_i:=E_Cylinder.OpenLockPush;
G_arrCylinder[_i].stInput.bHome:=GVL.I.bOpenLockPush_Cyl_H;
G_arrCylinder[_i].stInput.bWork:=GVL.I.bOpenLockPush_Cyl_W;
GVL.Q.bOpenLockPush_Cyl_H:=G_arrCylinder[_i].stOutput.bHome;
GVL.Q.bOpenLockPush_Cyl_W:=G_arrCylinder[_i].stOutput.bWork;

_i:=E_Cylinder.OpenLockRotate;
G_arrCylinder[_i].stInput.bHome:=GVL.I.bOpenLockRotate_Cyl_H;
G_arrCylinder[_i].stInput.bWork:=GVL.I.bOpenLockRotate_Cyl_W;
GVL.Q.bOpenLockRotate_Cyl_H:=G_arrCylinder[_i].stOutput.bHome;
GVL.Q.bOpenLockRotate_Cyl_W:=G_arrCylinder[_i].stOutput.bWork;

_i:=E_Cylinder.OpenLockPush2;
//G_arrCylinder[_i].stInput.bHome:=GVL.I.bOpenLockPush2_Cyl_H;
G_arrCylinder[_i].stInput.bHome:=NOT GVL.I.bOpenLockPush2_Cyl_W;
G_arrCylinder[_i].stInput.bWork:=GVL.I.bOpenLockPush2_Cyl_W;
GVL.Q.bOpenLockPush2_Cyl_H:=G_arrCylinder[_i].stOutput.bHome;
GVL.Q.bOpenLockPush2_Cyl_W:=G_arrCylinder[_i].stOutput.bWork;

_i:=E_Cylinder.TakeUcPrevent;
G_arrCylinder[_i].stInput.bWork:=GVL.I.bTakeUcPrevent_Cyl_W;
GVL.Q.bTakeUcPrevent_Cyl_H:=G_arrCylinder[_i].stOutput.bHome;
GVL.Q.bTakeUcPrevent_Cyl_W:=G_arrCylinder[_i].stOutput.bWork;

_i:=E_Cylinder.TakeUcLift;
G_arrCylinder[_i].stInput.bHome:=GVL.I.bTakeUcLift_Cyl_H;
G_arrCylinder[_i].stInput.bWork:=G_arrCylinder[_i].stOutput.bWork;//GVL.I.bTakeUcLift_Cyl_W;
GVL.Q.bTakeUcLift_Cyl_H:=G_arrCylinder[_i].stOutput.bHome;
GVL.Q.bTakeUcLift_Cyl_W:=G_arrCylinder[_i].stOutput.bWork;

_i:=E_Cylinder.TakeUcPush;
G_arrCylinder[_i].stInput.bHome:=GVL.I.bTakeUcPush_Cyl_H;
G_arrCylinder[_i].stInput.bWork:=GVL.I.bTakeUcPush_Cyl_W;
GVL.Q.bTakeUcPush_Cyl_H:=G_arrCylinder[_i].stOutput.bHome;
GVL.Q.bTakeUcPush_Cyl_W:=G_arrCylinder[_i].stOutput.bWork;

_i:=E_Cylinder.TakeUcRotate;
G_arrCylinder[_i].stInput.bHome:=GVL.I.bTakeUcRotate_Cyl_H;
G_arrCylinder[_i].stInput.bWork:=GVL.I.bTakeUcRotate_Cyl_W;
GVL.Q.bTakeUcRotate_Cyl_H:=G_arrCylinder[_i].stOutput.bHome;
GVL.Q.bTakeUcRotate_Cyl_W:=G_arrCylinder[_i].stOutput.bWork;

_i:=E_Cylinder.TakeUcStandard;
G_arrCylinder[_i].stInput.bHome:=GVL.I.bTakeUcStandard_Cyl_H;
G_arrCylinder[_i].stInput.bWork:=GVL.I.bTakeUcStandard_Cyl_W;
GVL.Q.bTakeUcStandard_Cyl_H:=G_arrCylinder[_i].stOutput.bHome;
GVL.Q.bTakeUcStandard_Cyl_W:=G_arrCylinder[_i].stOutput.bWork;

_i:=E_Cylinder.UnloadFrockPrevent;
G_arrCylinder[_i].stInput.bHome:=GVL.I.bUnloadFrockPrevent_Cyl_H;
G_arrCylinder[_i].stInput.bWork:=GVL.I.bUnloadFrockPrevent_Cyl_W;
GVL.Q.bUnloadFrockPrevent_Cyl_H:=G_arrCylinder[_i].stOutput.bHome;
GVL.Q.bUnloadFrockPrevent_Cyl_W:=G_arrCylinder[_i].stOutput.bWork;

_i:=E_Cylinder.UnloadFrockLift;
G_arrCylinder[_i].stInput.bHome:=GVL.I.bUnloadFrockLift_Cyl_H;
G_arrCylinder[_i].stInput.bWork:=GVL.I.bUnloadFrockLift_Cyl_W;
GVL.Q.bUnloadFrockLift_Cyl_H:=G_arrCylinder[_i].stOutput.bHome;
GVL.Q.bUnloadFrockLift_Cyl_W:=G_arrCylinder[_i].stOutput.bWork;

_i:=E_Cylinder.UnloadFrockPush;
G_arrCylinder[_i].stInput.bHome:=GVL.I.bUnloadFrockPush_Cyl_H;
G_arrCylinder[_i].stInput.bWork:=GVL.I.bUnloadFrockPush_Cyl_W;
GVL.Q.bUnloadFrockPush_Cyl_H:=G_arrCylinder[_i].stOutput.bHome;
GVL.Q.bUnloadFrockPush_Cyl_W:=G_arrCylinder[_i].stOutput.bWork;

_i:=E_Cylinder.TakeUc1Y;
G_arrCylinder[_i].stInput.bHome:=GVL.I.bTakeUc1Y_Cyl_H;
G_arrCylinder[_i].stInput.bWork:=GVL.I.bTakeUc1Y_Cyl_W;
GVL.Q.bTakeUc1Y_Cyl_H:=G_arrCylinder[_i].stOutput.bHome;
GVL.Q.bTakeUc1Y_Cyl_W:=G_arrCylinder[_i].stOutput.bWork;

_i:=E_Cylinder.TakeUc1Z1;
G_arrCylinder[_i].stInput.bHome:=GVL.I.bTakeUc1Z1_Cyl_H;
G_arrCylinder[_i].stInput.bWork:=GVL.I.bTakeUc1Z1_Cyl_W;
GVL.Q.bTakeUc1Z1_Cyl_H:=G_arrCylinder[_i].stOutput.bHome;
GVL.Q.bTakeUc1Z1_Cyl_W:=G_arrCylinder[_i].stOutput.bWork;

_i:=E_Cylinder.TakeUc1Z2;
G_arrCylinder[_i].stInput.bHome:=GVL.I.bTakeUc1Z2_Cyl_H;
G_arrCylinder[_i].stInput.bWork:=GVL.I.bTakeUc1Z2_Cyl_W;
GVL.Q.bTakeUc1Z2_Cyl_H:=G_arrCylinder[_i].stOutput.bHome;
GVL.Q.bTakeUc1Z2_Cyl_W:=G_arrCylinder[_i].stOutput.bWork;

_i:=E_Cylinder.TakeUc1Rotate;
G_arrCylinder[_i].stInput.bHome:=GVL.I.bTakeUc1Rotate_Cyl_H;
G_arrCylinder[_i].stInput.bWork:=GVL.I.bTakeUc1Rotate_Cyl_W;
GVL.Q.bTakeUc1Rotate_Cyl_H:=G_arrCylinder[_i].stOutput.bHome;
GVL.Q.bTakeUc1Rotate_Cyl_W:=G_arrCylinder[_i].stOutput.bWork;

_i:=E_Cylinder.TakeUc1Clamp;
G_arrCylinder[_i].stInput.bHome:=GVL.I.bTakeUc1Clamp_Cyl_H;
//G_arrCylinder[_i].stInput.bWork:=GVL.I.bTakeUc1Clamp_Cyl_W;
GVL.Q.bTakeUc1Clamp_Cyl_H:=G_arrCylinder[_i].stOutput.bHome;
GVL.Q.bTakeUc1Clamp_Cyl_W:=G_arrCylinder[_i].stOutput.bWork;

_i:=E_Cylinder.UnloadUcElevator;
//G_arrCylinder[_i].stInput.bHome:=GVL.I.bUnloadUcElevator_Cyl_H;
//G_arrCylinder[_i].stInput.bWork:=GVL.I.bUnloadUcElevator_Cyl_W;
GVL.Q.bUnloadUcElevator_Cyl_H:=G_arrCylinder[_i].stOutput.bHome;
GVL.Q.bUnloadUcElevator_Cyl_W:=G_arrCylinder[_i].stOutput.bWork;

_i:=E_Cylinder.UnloadUcConveyorPush;
//G_arrCylinder[_i].stInput.bHome:=GVL.I.bUnloadUcConveyorPush_Cyl_H;
//G_arrCylinder[_i].stInput.bWork:=GVL.I.bUnloadUcConveyorPush_Cyl_W;
GVL.Q.bUnloadUcConveyorPush_Cyl_H:=G_arrCylinder[_i].stOutput.bHome;
GVL.Q.bUnloadUcConveyorPush_Cyl_W:=G_arrCylinder[_i].stOutput.bWork;

_i:=E_Cylinder.UnloadFrockConveyorPrevent;
//G_arrCylinder[_i].stInput.bHome:=GVL.I.bUnloadFrockConveyorPrevent_Cyl_H;
//G_arrCylinder[_i].stInput.bWork:=GVL.I.bUnloadFrockConveyorPrevent_Cyl_W;
GVL.Q.bUnloadFrockConveyorPrevent_Cyl_H:=G_arrCylinder[_i].stOutput.bHome;
GVL.Q.bUnloadFrockConveyorPrevent_Cyl_W:=G_arrCylinder[_i].stOutput.bWork;

_i:=E_Cylinder.UnloadFrockConveyorPush;
//G_arrCylinder[_i].stInput.bHome:=GVL.I.bUnloadFrockConveyorPush_Cyl_H;
//G_arrCylinder[_i].stInput.bWork:=GVL.I.bUnloadFrockConveyorPush_Cyl_W;
GVL.Q.bUnloadFrockConveyorPush_Cyl_H:=G_arrCylinder[_i].stOutput.bHome;
GVL.Q.bUnloadFrockConveyorPush_Cyl_W:=G_arrCylinder[_i].stOutput.bWork;

_i:=E_Cylinder.OpenLockElevator;
G_arrCylinder[_i].stInput.bHome:=GVL.I.bOpenLockElevator_Cyl_H;
G_arrCylinder[_i].stInput.bWork:=GVL.I.bOpenLockElevator_Cyl_W;
GVL.Q.bOpenLockElevator_Cyl_H:=G_arrCylinder[_i].stOutput.bHome;
GVL.Q.bOpenLockElevator_Cyl_W:=G_arrCylinder[_i].stOutput.bWork;

_i:=E_Cylinder.OpenLockPin;
G_arrCylinder[_i].stInput.bWork:=G_arrCylinder[_i].stOutput.bWork;//GVL.I.bOpenLockPin_Cyl_W;
GVL.Q.bOpenLockPin_Cyl_H:=G_arrCylinder[_i].stOutput.bHome;
GVL.Q.bOpenLockPin_Cyl_W:=G_arrCylinder[_i].stOutput.bWork;

_i:=E_Cylinder.TakeUcElevator;
G_arrCylinder[_i].stInput.bHome:=GVL.I.bTakeUcElevator_Cyl_H;
G_arrCylinder[_i].stInput.bWork:=GVL.I.bTakeUcElevator_Cyl_W;
GVL.Q.bTakeUcElevator_Cyl_H:=G_arrCylinder[_i].stOutput.bHome;
GVL.Q.bTakeUcElevator_Cyl_W:=G_arrCylinder[_i].stOutput.bWork;

_i:=E_Cylinder.TakeUcPush1;
G_arrCylinder[_i].stInput.bHome:=GVL.I.bTakeUcPush1_Cyl_H;
G_arrCylinder[_i].stInput.bWork:=GVL.I.bTakeUcPush1_Cyl_W;
GVL.Q.bTakeUcPush1_Cyl_H:=G_arrCylinder[_i].stOutput.bHome;
GVL.Q.bTakeUcPush1_Cyl_W:=G_arrCylinder[_i].stOutput.bWork;

_i:=E_Cylinder.UnloadUcBeltTipper;
G_arrCylinder[_i].stInput.bHome:=GVL.I.bUnloadUcBeltTipper_Cyl_H;
G_arrCylinder[_i].stInput.bWork:=GVL.I.bUnloadUcBeltTipper_Cyl_W;
GVL.Q.bUnloadUcBeltTipper_Cyl_H:=G_arrCylinder[_i].stOutput.bHome;
GVL.Q.bUnloadUcBeltTipper_Cyl_W:=G_arrCylinder[_i].stOutput.bWork;

_i:=E_Cylinder.UnloadUcBeltLift;
G_arrCylinder[_i].stInput.bHome:=GVL.I.bUnloadUcBeltLift_Cyl_H;
G_arrCylinder[_i].stInput.bWork:=GVL.I.bUnloadUcBeltLift_Cyl_W;
GVL.Q.bUnloadUcBeltLift_Cyl_H:=G_arrCylinder[_i].stOutput.bHome;
GVL.Q.bUnloadUcBeltLift_Cyl_W:=G_arrCylinder[_i].stOutput.bWork;

_i:=E_Cylinder.OpenLockTranslation;
G_arrCylinder[_i].stInput.bHome:=GVL.I.bOpenLockTranslation_Cyl_H;
G_arrCylinder[_i].stInput.bWork:=GVL.I.bOpenLockTranslation_Cyl_W;
GVL.Q.bOpenLockTranslation_Cyl_H:=G_arrCylinder[_i].stOutput.bHome;
GVL.Q.bOpenLockTranslation_Cyl_W:=G_arrCylinder[_i].stOutput.bWork;

_i:=E_Cylinder.TakeUcFrockClamp;
G_arrCylinder[_i].stInput.bHome:=GVL.I.bTakeUcFrockClamp_Cyl_H;
G_arrCylinder[_i].stInput.bWork:=GVL.I.bTakeUcFrockClamp_Cyl_W;
GVL.Q.bTakeUcFrockClamp_Cyl_H:=G_arrCylinder[_i].stOutput.bHome;
GVL.Q.bTakeUcFrockClamp_Cyl_W:=G_arrCylinder[_i].stOutput.bWork;
END_ACTION

ACTION A_CylinderTest367:
FOR _i:=0 TO 50 BY 1 DO
	G_arrCylinder[_i].ID:=TO_BYTE(_i+50);
	_arrCylTon_H[_i](IN:=G_arrCylinder[_i].stOutput.bHome , PT:=T#2S , Q=> , ET=> );
	_arrCylTon_W[_i](IN:=G_arrCylinder[_i].stOutput.bWork , PT:=T#2S , Q=> , ET=> );
	G_arrCylinder[_i].stInput.bHome:=_arrCylTon_H[_i].Q;
	G_arrCylinder[_i].stInput.bWork:=_arrCylTon_W[_i].Q;
END_FOR

_i:=E_Cylinder.Line0Part;
GVL.Q.bLine0Part_Cyl_H:=G_arrCylinder[_i].stOutput.bHome;
GVL.Q.bLine0Part_Cyl_W:=G_arrCylinder[_i].stOutput.bWork;

_i:=E_Cylinder.Line0Prevent;
GVL.Q.bLine0Prevent_Cyl_H:=G_arrCylinder[_i].stOutput.bHome;
GVL.Q.bLine0Prevent_Cyl_W:=G_arrCylinder[_i].stOutput.bWork;

_i:=E_Cylinder.Line0Push;
G_arrCylinder[_i].stInput.bHome:=GVL.I.bLine0Push_Cyl_H;
G_arrCylinder[_i].stInput.bWork:=GVL.I.bLine0Push_Cyl_W;
GVL.Q.bLine0Push_Cyl_H:=G_arrCylinder[_i].stOutput.bHome;
GVL.Q.bLine0Push_Cyl_W:=G_arrCylinder[_i].stOutput.bWork;

_i:=E_Cylinder.AcquirePrevent0;
G_arrCylinder[_i].stInput.bWork:=GVL.I.bAcquirePrevent0_Cyl_W;
GVL.Q.bAcquirePrevent0_Cyl_H:=G_arrCylinder[_i].stOutput.bHome;
GVL.Q.bAcquirePrevent0_Cyl_W:=G_arrCylinder[_i].stOutput.bWork;

_i:=E_Cylinder.AcquirePrevent1;
G_arrCylinder[_i].stInput.bWork:=GVL.I.bAcquirePrevent1_Cyl_W;
GVL.Q.bAcquirePrevent1_Cyl_H:=G_arrCylinder[_i].stOutput.bHome;
GVL.Q.bAcquirePrevent1_Cyl_W:=G_arrCylinder[_i].stOutput.bWork;

_i:=E_Cylinder.AcquireLift;
G_arrCylinder[_i].stInput.bHome:=GVL.I.bAcquireLift_Cyl_H;
G_arrCylinder[_i].stInput.bWork:=GVL.I.bAcquireLift_Cyl_W;
GVL.Q.bAcquireLift_Cyl_H:=G_arrCylinder[_i].stOutput.bHome;
GVL.Q.bAcquireLift_Cyl_W:=G_arrCylinder[_i].stOutput.bWork;

_i:=E_Cylinder.AcquirePush;
G_arrCylinder[_i].stInput.bHome:=GVL.I.bAcquirePush_Cyl_H;
G_arrCylinder[_i].stInput.bWork:=GVL.I.bAcquirePush_Cyl_W;
GVL.Q.bAcquirePush_Cyl_H:=G_arrCylinder[_i].stOutput.bHome;
GVL.Q.bAcquirePush_Cyl_W:=G_arrCylinder[_i].stOutput.bWork;

_i:=E_Cylinder.AcquireElevator;
G_arrCylinder[_i].stInput.bHome:=GVL.I.bAcquireElevator_Cyl_H;
G_arrCylinder[_i].stInput.bWork:=GVL.I.bAcquireElevator_Cyl_W;
GVL.Q.bAcquireElevator_Cyl_H:=G_arrCylinder[_i].stOutput.bHome;
GVL.Q.bAcquireElevator_Cyl_W:=G_arrCylinder[_i].stOutput.bWork;

_i:=E_Cylinder.SteeringLift;
G_arrCylinder[_i].stInput.bHome:=GVL.I.bSteeringLift_Cyl_H;
G_arrCylinder[_i].stInput.bWork:=GVL.I.bSteeringLift_Cyl_W;
GVL.Q.bSteeringLift_Cyl_H:=G_arrCylinder[_i].stOutput.bHome;
GVL.Q.bSteeringLift_Cyl_W:=G_arrCylinder[_i].stOutput.bWork;

_i:=E_Cylinder.SteeringAcquireElevator;
G_arrCylinder[_i].stInput.bHome:=GVL.I.bSteeringAcquireElevator_Cyl_H;
G_arrCylinder[_i].stInput.bWork:=GVL.I.bSteeringAcquireElevator_Cyl_W;
GVL.Q.bSteeringAcquireElevator_Cyl_H:=G_arrCylinder[_i].stOutput.bHome;
GVL.Q.bSteeringAcquireElevator_Cyl_W:=G_arrCylinder[_i].stOutput.bWork;

_i:=E_Cylinder.SteeringRotate;
G_arrCylinder[_i].stInput.bHome:=GVL.I.bSteeringRotate_Cyl_H;
G_arrCylinder[_i].stInput.bWork:=GVL.I.bSteeringRotate_Cyl_W;
GVL.Q.bSteeringRotate_Cyl_H:=G_arrCylinder[_i].stOutput.bHome;
GVL.Q.bSteeringRotate_Cyl_W:=G_arrCylinder[_i].stOutput.bWork;

_i:=E_Cylinder.SteeringAcquireLimit;
G_arrCylinder[_i].stInput.bHome:=GVL.I.bSteeringAcquireLimit_Cyl_H;
G_arrCylinder[_i].stInput.bWork:=GVL.I.bSteeringAcquireLimit_Cyl_W;
GVL.Q.bSteeringAcquireLimit_Cyl_H:=G_arrCylinder[_i].stOutput.bHome;
GVL.Q.bSteeringAcquireLimit_Cyl_W:=G_arrCylinder[_i].stOutput.bWork;

_i:=E_Cylinder.OpenLockPrevent;
G_arrCylinder[_i].stInput.bWork:=GVL.I.bOpenLockPrevent_Cyl_W;
GVL.Q.bOpenLockPrevent_Cyl_H:=G_arrCylinder[_i].stOutput.bHome;
GVL.Q.bOpenLockPrevent_Cyl_W:=G_arrCylinder[_i].stOutput.bWork;

_i:=E_Cylinder.OpenLockLift;
G_arrCylinder[_i].stInput.bHome:=GVL.I.bOpenLockLift_Cyl_H;
G_arrCylinder[_i].stInput.bWork:=GVL.I.bOpenLockLift_Cyl_W;
GVL.Q.bOpenLockLift_Cyl_H:=G_arrCylinder[_i].stOutput.bHome;
GVL.Q.bOpenLockLift_Cyl_W:=G_arrCylinder[_i].stOutput.bWork;

_i:=E_Cylinder.OpenLockPush;
G_arrCylinder[_i].stInput.bHome:=GVL.I.bOpenLockPush_Cyl_H;
G_arrCylinder[_i].stInput.bWork:=GVL.I.bOpenLockPush_Cyl_W;
GVL.Q.bOpenLockPush_Cyl_H:=G_arrCylinder[_i].stOutput.bHome;
GVL.Q.bOpenLockPush_Cyl_W:=G_arrCylinder[_i].stOutput.bWork;

_i:=E_Cylinder.OpenLockRotate;
G_arrCylinder[_i].stInput.bHome:=GVL.I.bOpenLockRotate_Cyl_H;
G_arrCylinder[_i].stInput.bWork:=GVL.I.bOpenLockRotate_Cyl_W;
GVL.Q.bOpenLockRotate_Cyl_H:=G_arrCylinder[_i].stOutput.bHome;
GVL.Q.bOpenLockRotate_Cyl_W:=G_arrCylinder[_i].stOutput.bWork;

_i:=E_Cylinder.OpenLockPush2;
//G_arrCylinder[_i].stInput.bHome:=GVL.I.bOpenLockPush2_Cyl_H;
G_arrCylinder[_i].stInput.bHome:=NOT GVL.I.bOpenLockPush2_Cyl_W;
G_arrCylinder[_i].stInput.bWork:=GVL.I.bOpenLockPush2_Cyl_W;
GVL.Q.bOpenLockPush2_Cyl_H:=G_arrCylinder[_i].stOutput.bHome;
GVL.Q.bOpenLockPush2_Cyl_W:=G_arrCylinder[_i].stOutput.bWork;

_i:=E_Cylinder.TakeUcPrevent;
G_arrCylinder[_i].stInput.bWork:=GVL.I.bTakeUcPrevent_Cyl_W;
GVL.Q.bTakeUcPrevent_Cyl_H:=G_arrCylinder[_i].stOutput.bHome;
GVL.Q.bTakeUcPrevent_Cyl_W:=G_arrCylinder[_i].stOutput.bWork;

_i:=E_Cylinder.TakeUcLift;
G_arrCylinder[_i].stInput.bHome:=GVL.I.bTakeUcLift_Cyl_H;
G_arrCylinder[_i].stInput.bWork:=GVL.I.bTakeUcLift_Cyl_W;
GVL.Q.bTakeUcLift_Cyl_H:=G_arrCylinder[_i].stOutput.bHome;
GVL.Q.bTakeUcLift_Cyl_W:=G_arrCylinder[_i].stOutput.bWork;

_i:=E_Cylinder.TakeUcPush;
G_arrCylinder[_i].stInput.bHome:=GVL.I.bTakeUcPush_Cyl_H;
G_arrCylinder[_i].stInput.bWork:=GVL.I.bTakeUcPush_Cyl_W;
GVL.Q.bTakeUcPush_Cyl_H:=G_arrCylinder[_i].stOutput.bHome;
GVL.Q.bTakeUcPush_Cyl_W:=G_arrCylinder[_i].stOutput.bWork;

_i:=E_Cylinder.TakeUcRotate;
G_arrCylinder[_i].stInput.bHome:=GVL.I.bTakeUcRotate_Cyl_H;
G_arrCylinder[_i].stInput.bWork:=GVL.I.bTakeUcRotate_Cyl_W;
GVL.Q.bTakeUcRotate_Cyl_H:=G_arrCylinder[_i].stOutput.bHome;
GVL.Q.bTakeUcRotate_Cyl_W:=G_arrCylinder[_i].stOutput.bWork;

_i:=E_Cylinder.TakeUcStandard;
G_arrCylinder[_i].stInput.bHome:=GVL.I.bTakeUcStandard_Cyl_H;
G_arrCylinder[_i].stInput.bWork:=GVL.I.bTakeUcStandard_Cyl_W;
GVL.Q.bTakeUcStandard_Cyl_H:=G_arrCylinder[_i].stOutput.bHome;
GVL.Q.bTakeUcStandard_Cyl_W:=G_arrCylinder[_i].stOutput.bWork;

_i:=E_Cylinder.UnloadFrockPrevent;
G_arrCylinder[_i].stInput.bHome:=GVL.I.bUnloadFrockPrevent_Cyl_H;
G_arrCylinder[_i].stInput.bWork:=GVL.I.bUnloadFrockPrevent_Cyl_W;
GVL.Q.bUnloadFrockPrevent_Cyl_H:=G_arrCylinder[_i].stOutput.bHome;
GVL.Q.bUnloadFrockPrevent_Cyl_W:=G_arrCylinder[_i].stOutput.bWork;

_i:=E_Cylinder.UnloadFrockLift;
G_arrCylinder[_i].stInput.bHome:=GVL.I.bUnloadFrockLift_Cyl_H;
G_arrCylinder[_i].stInput.bWork:=GVL.I.bUnloadFrockLift_Cyl_W;
GVL.Q.bUnloadFrockLift_Cyl_H:=G_arrCylinder[_i].stOutput.bHome;
GVL.Q.bUnloadFrockLift_Cyl_W:=G_arrCylinder[_i].stOutput.bWork;

_i:=E_Cylinder.UnloadFrockPush;
G_arrCylinder[_i].stInput.bHome:=GVL.I.bUnloadFrockPush_Cyl_H;
G_arrCylinder[_i].stInput.bWork:=GVL.I.bUnloadFrockPush_Cyl_W;
GVL.Q.bUnloadFrockPush_Cyl_H:=G_arrCylinder[_i].stOutput.bHome;
GVL.Q.bUnloadFrockPush_Cyl_W:=G_arrCylinder[_i].stOutput.bWork;

_i:=E_Cylinder.TakeUc1Y;
G_arrCylinder[_i].stInput.bHome:=GVL.I.bTakeUc1Y_Cyl_H;
G_arrCylinder[_i].stInput.bWork:=GVL.I.bTakeUc1Y_Cyl_W;
GVL.Q.bTakeUc1Y_Cyl_H:=G_arrCylinder[_i].stOutput.bHome;
GVL.Q.bTakeUc1Y_Cyl_W:=G_arrCylinder[_i].stOutput.bWork;

_i:=E_Cylinder.TakeUc1Z1;
G_arrCylinder[_i].stInput.bHome:=GVL.I.bTakeUc1Z1_Cyl_H;
G_arrCylinder[_i].stInput.bWork:=GVL.I.bTakeUc1Z1_Cyl_W;
GVL.Q.bTakeUc1Z1_Cyl_H:=G_arrCylinder[_i].stOutput.bHome;
GVL.Q.bTakeUc1Z1_Cyl_W:=G_arrCylinder[_i].stOutput.bWork;

_i:=E_Cylinder.TakeUc1Z2;
G_arrCylinder[_i].stInput.bHome:=GVL.I.bTakeUc1Z2_Cyl_H;
G_arrCylinder[_i].stInput.bWork:=GVL.I.bTakeUc1Z2_Cyl_W;
GVL.Q.bTakeUc1Z2_Cyl_H:=G_arrCylinder[_i].stOutput.bHome;
GVL.Q.bTakeUc1Z2_Cyl_W:=G_arrCylinder[_i].stOutput.bWork;

_i:=E_Cylinder.TakeUc1Rotate;
G_arrCylinder[_i].stInput.bHome:=GVL.I.bTakeUc1Rotate_Cyl_H;
G_arrCylinder[_i].stInput.bWork:=GVL.I.bTakeUc1Rotate_Cyl_W;
GVL.Q.bTakeUc1Rotate_Cyl_H:=G_arrCylinder[_i].stOutput.bHome;
GVL.Q.bTakeUc1Rotate_Cyl_W:=G_arrCylinder[_i].stOutput.bWork;

_i:=E_Cylinder.TakeUc1Clamp;
G_arrCylinder[_i].stInput.bHome:=GVL.I.bTakeUc1Clamp_Cyl_H;
//G_arrCylinder[_i].stInput.bWork:=GVL.I.bTakeUc1Clamp_Cyl_W;
GVL.Q.bTakeUc1Clamp_Cyl_H:=G_arrCylinder[_i].stOutput.bHome;
GVL.Q.bTakeUc1Clamp_Cyl_W:=G_arrCylinder[_i].stOutput.bWork;

_i:=E_Cylinder.UnloadUcElevator;
//G_arrCylinder[_i].stInput.bHome:=GVL.I.bUnloadUcElevator_Cyl_H;
//G_arrCylinder[_i].stInput.bWork:=GVL.I.bUnloadUcElevator_Cyl_W;
GVL.Q.bUnloadUcElevator_Cyl_H:=G_arrCylinder[_i].stOutput.bHome;
GVL.Q.bUnloadUcElevator_Cyl_W:=G_arrCylinder[_i].stOutput.bWork;

_i:=E_Cylinder.UnloadUcConveyorPush;
//G_arrCylinder[_i].stInput.bHome:=GVL.I.bUnloadUcConveyorPush_Cyl_H;
//G_arrCylinder[_i].stInput.bWork:=GVL.I.bUnloadUcConveyorPush_Cyl_W;
GVL.Q.bUnloadUcConveyorPush_Cyl_H:=G_arrCylinder[_i].stOutput.bHome;
GVL.Q.bUnloadUcConveyorPush_Cyl_W:=G_arrCylinder[_i].stOutput.bWork;

_i:=E_Cylinder.UnloadFrockConveyorPrevent;
//G_arrCylinder[_i].stInput.bHome:=GVL.I.bUnloadFrockConveyorPrevent_Cyl_H;
//G_arrCylinder[_i].stInput.bWork:=GVL.I.bUnloadFrockConveyorPrevent_Cyl_W;
GVL.Q.bUnloadFrockConveyorPrevent_Cyl_H:=G_arrCylinder[_i].stOutput.bHome;
GVL.Q.bUnloadFrockConveyorPrevent_Cyl_W:=G_arrCylinder[_i].stOutput.bWork;

_i:=E_Cylinder.UnloadFrockConveyorPush;
//G_arrCylinder[_i].stInput.bHome:=GVL.I.bUnloadFrockConveyorPush_Cyl_H;
//G_arrCylinder[_i].stInput.bWork:=GVL.I.bUnloadFrockConveyorPush_Cyl_W;
GVL.Q.bUnloadFrockConveyorPush_Cyl_H:=G_arrCylinder[_i].stOutput.bHome;
GVL.Q.bUnloadFrockConveyorPush_Cyl_W:=G_arrCylinder[_i].stOutput.bWork;

_i:=E_Cylinder.OpenLockElevator;
G_arrCylinder[_i].stInput.bHome:=GVL.I.bOpenLockElevator_Cyl_H;
G_arrCylinder[_i].stInput.bWork:=GVL.I.bOpenLockElevator_Cyl_W;
GVL.Q.bOpenLockElevator_Cyl_H:=G_arrCylinder[_i].stOutput.bHome;
GVL.Q.bOpenLockElevator_Cyl_W:=G_arrCylinder[_i].stOutput.bWork;

_i:=E_Cylinder.OpenLockPin;
G_arrCylinder[_i].stInput.bHome:=GVL.I.bOpenLockPin_Cyl_H;
G_arrCylinder[_i].stInput.bWork:=GVL.I.bOpenLockPin_Cyl_W;
GVL.Q.bOpenLockPin_Cyl_H:=G_arrCylinder[_i].stOutput.bHome;
GVL.Q.bOpenLockPin_Cyl_W:=G_arrCylinder[_i].stOutput.bWork;

_i:=E_Cylinder.TakeUcElevator;
G_arrCylinder[_i].stInput.bHome:=GVL.I.bTakeUcElevator_Cyl_H;
G_arrCylinder[_i].stInput.bWork:=GVL.I.bTakeUcElevator_Cyl_W;
GVL.Q.bTakeUcElevator_Cyl_H:=G_arrCylinder[_i].stOutput.bHome;
GVL.Q.bTakeUcElevator_Cyl_W:=G_arrCylinder[_i].stOutput.bWork;

_i:=E_Cylinder.TakeUcPush1;
G_arrCylinder[_i].stInput.bHome:=GVL.I.bTakeUcPush1_Cyl_H;
G_arrCylinder[_i].stInput.bWork:=GVL.I.bTakeUcPush1_Cyl_W;
GVL.Q.bTakeUcPush1_Cyl_H:=G_arrCylinder[_i].stOutput.bHome;
GVL.Q.bTakeUcPush1_Cyl_W:=G_arrCylinder[_i].stOutput.bWork;

_i:=E_Cylinder.UnloadUcBeltTipper;
G_arrCylinder[_i].stInput.bHome:=GVL.I.bUnloadUcBeltTipper_Cyl_H;
G_arrCylinder[_i].stInput.bWork:=GVL.I.bUnloadUcBeltTipper_Cyl_W;
GVL.Q.bUnloadUcBeltTipper_Cyl_H:=G_arrCylinder[_i].stOutput.bHome;
GVL.Q.bUnloadUcBeltTipper_Cyl_W:=G_arrCylinder[_i].stOutput.bWork;

_i:=E_Cylinder.UnloadUcBeltLift;
G_arrCylinder[_i].stInput.bHome:=GVL.I.bUnloadUcBeltLift_Cyl_H;
G_arrCylinder[_i].stInput.bWork:=GVL.I.bUnloadUcBeltLift_Cyl_W;
GVL.Q.bUnloadUcBeltLift_Cyl_H:=G_arrCylinder[_i].stOutput.bHome;
GVL.Q.bUnloadUcBeltLift_Cyl_W:=G_arrCylinder[_i].stOutput.bWork;

_i:=E_Cylinder.OpenLockTranslation;
G_arrCylinder[_i].stInput.bHome:=GVL.I.bOpenLockTranslation_Cyl_H;
G_arrCylinder[_i].stInput.bWork:=GVL.I.bOpenLockTranslation_Cyl_W;
GVL.Q.bOpenLockTranslation_Cyl_H:=G_arrCylinder[_i].stOutput.bHome;
GVL.Q.bOpenLockTranslation_Cyl_W:=G_arrCylinder[_i].stOutput.bWork;

_i:=E_Cylinder.TakeUcFrockClamp;
G_arrCylinder[_i].stInput.bHome:=G_arrCylinder[_i].stOutput.bHome;
G_arrCylinder[_i].stInput.bWork:=G_arrCylinder[_i].stOutput.bWork;
GVL.Q.bTakeUcFrockClamp_Cyl_H:=G_arrCylinder[_i].stOutput.bHome;
GVL.Q.bTakeUcFrockClamp_Cyl_W:=G_arrCylinder[_i].stOutput.bWork;
END_ACTION

ACTION A_CylinderTest373:
FOR _i:=0 TO 50 BY 1 DO
	G_arrCylinder[_i].ID:=TO_BYTE(_i+50);
	_arrCylTon_H[_i](IN:=G_arrCylinder[_i].stOutput.bHome , PT:=T#2S , Q=> , ET=> );
	_arrCylTon_W[_i](IN:=G_arrCylinder[_i].stOutput.bWork , PT:=T#2S , Q=> , ET=> );
	G_arrCylinder[_i].stInput.bHome:=_arrCylTon_H[_i].Q;
	G_arrCylinder[_i].stInput.bWork:=_arrCylTon_W[_i].Q;
END_FOR

_i:=E_Cylinder.Line0Part;
GVL.Q.bLine0Part_Cyl_H:=G_arrCylinder[_i].stOutput.bHome;
GVL.Q.bLine0Part_Cyl_W:=G_arrCylinder[_i].stOutput.bWork;

_i:=E_Cylinder.Line0Prevent;
GVL.Q.bLine0Prevent_Cyl_H:=G_arrCylinder[_i].stOutput.bHome;
GVL.Q.bLine0Prevent_Cyl_W:=G_arrCylinder[_i].stOutput.bWork;

_i:=E_Cylinder.Line0Push;
GVL.Q.bLine0Push_Cyl_H:=G_arrCylinder[_i].stOutput.bHome;
GVL.Q.bLine0Push_Cyl_W:=G_arrCylinder[_i].stOutput.bWork;

_i:=E_Cylinder.AcquirePrevent0;
G_arrCylinder[_i].stInput.bWork:=GVL.I.bAcquirePrevent0_Cyl_W;
GVL.Q.bAcquirePrevent0_Cyl_H:=G_arrCylinder[_i].stOutput.bHome;
GVL.Q.bAcquirePrevent0_Cyl_W:=G_arrCylinder[_i].stOutput.bWork;

_i:=E_Cylinder.AcquirePrevent1;
G_arrCylinder[_i].stInput.bWork:=GVL.I.bAcquirePrevent1_Cyl_W;
GVL.Q.bAcquirePrevent1_Cyl_H:=G_arrCylinder[_i].stOutput.bHome;
GVL.Q.bAcquirePrevent1_Cyl_W:=G_arrCylinder[_i].stOutput.bWork;

_i:=E_Cylinder.AcquireLift;
G_arrCylinder[_i].stInput.bHome:=GVL.I.bAcquireLift_Cyl_H;
G_arrCylinder[_i].stInput.bWork:=GVL.I.bAcquireLift_Cyl_W;
GVL.Q.bAcquireLift_Cyl_H:=G_arrCylinder[_i].stOutput.bHome;
GVL.Q.bAcquireLift_Cyl_W:=G_arrCylinder[_i].stOutput.bWork;

_i:=E_Cylinder.AcquirePush;
G_arrCylinder[_i].stInput.bHome:=GVL.I.bAcquirePush_Cyl_H;
G_arrCylinder[_i].stInput.bWork:=GVL.I.bAcquirePush_Cyl_W;
GVL.Q.bAcquirePush_Cyl_H:=G_arrCylinder[_i].stOutput.bHome;
GVL.Q.bAcquirePush_Cyl_W:=G_arrCylinder[_i].stOutput.bWork;

_i:=E_Cylinder.AcquireElevator;
G_arrCylinder[_i].stInput.bHome:=GVL.I.bAcquireElevator_Cyl_H;
G_arrCylinder[_i].stInput.bWork:=GVL.I.bAcquireElevator_Cyl_W;
GVL.Q.bAcquireElevator_Cyl_H:=G_arrCylinder[_i].stOutput.bHome;
GVL.Q.bAcquireElevator_Cyl_W:=G_arrCylinder[_i].stOutput.bWork;

_i:=E_Cylinder.SteeringLift;
G_arrCylinder[_i].stInput.bHome:=GVL.I.bSteeringLift_Cyl_H;
G_arrCylinder[_i].stInput.bWork:=GVL.I.bSteeringLift_Cyl_W;
GVL.Q.bSteeringLift_Cyl_H:=G_arrCylinder[_i].stOutput.bHome;
GVL.Q.bSteeringLift_Cyl_W:=G_arrCylinder[_i].stOutput.bWork;

_i:=E_Cylinder.SteeringAcquireElevator;
G_arrCylinder[_i].stInput.bHome:=GVL.I.bSteeringAcquireElevator_Cyl_H;
G_arrCylinder[_i].stInput.bWork:=GVL.I.bSteeringAcquireElevator_Cyl_W;
GVL.Q.bSteeringAcquireElevator_Cyl_H:=G_arrCylinder[_i].stOutput.bHome;
GVL.Q.bSteeringAcquireElevator_Cyl_W:=G_arrCylinder[_i].stOutput.bWork;

_i:=E_Cylinder.SteeringRotate;
G_arrCylinder[_i].stInput.bHome:=GVL.I.bSteeringRotate_Cyl_H;
G_arrCylinder[_i].stInput.bWork:=GVL.I.bSteeringRotate_Cyl_W;
GVL.Q.bSteeringRotate_Cyl_H:=G_arrCylinder[_i].stOutput.bHome;
GVL.Q.bSteeringRotate_Cyl_W:=G_arrCylinder[_i].stOutput.bWork;

_i:=E_Cylinder.SteeringAcquireLimit;
G_arrCylinder[_i].stInput.bHome:=GVL.I.bSteeringAcquireLimit_Cyl_H;
G_arrCylinder[_i].stInput.bWork:=GVL.I.bSteeringAcquireLimit_Cyl_W;
GVL.Q.bSteeringAcquireLimit_Cyl_H:=G_arrCylinder[_i].stOutput.bHome;
GVL.Q.bSteeringAcquireLimit_Cyl_W:=G_arrCylinder[_i].stOutput.bWork;

_i:=E_Cylinder.OpenLockPrevent;
G_arrCylinder[_i].stInput.bWork:=GVL.I.bOpenLockPrevent_Cyl_W;
GVL.Q.bOpenLockPrevent_Cyl_H:=G_arrCylinder[_i].stOutput.bHome;
GVL.Q.bOpenLockPrevent_Cyl_W:=G_arrCylinder[_i].stOutput.bWork;

_i:=E_Cylinder.OpenLockLift;
G_arrCylinder[_i].stInput.bHome:=GVL.I.bOpenLockLift_Cyl_H;
G_arrCylinder[_i].stInput.bWork:=GVL.I.bOpenLockLift_Cyl_W;
GVL.Q.bOpenLockLift_Cyl_H:=G_arrCylinder[_i].stOutput.bHome;
GVL.Q.bOpenLockLift_Cyl_W:=G_arrCylinder[_i].stOutput.bWork;

_i:=E_Cylinder.OpenLockPush;
G_arrCylinder[_i].stInput.bHome:=GVL.I.bOpenLockPush_Cyl_H;
G_arrCylinder[_i].stInput.bWork:=GVL.I.bOpenLockPush_Cyl_W;
GVL.Q.bOpenLockPush_Cyl_H:=G_arrCylinder[_i].stOutput.bHome;
GVL.Q.bOpenLockPush_Cyl_W:=G_arrCylinder[_i].stOutput.bWork;

_i:=E_Cylinder.OpenLockRotate;
G_arrCylinder[_i].stInput.bHome:=GVL.I.bOpenLockRotate_Cyl_H;
G_arrCylinder[_i].stInput.bWork:=GVL.I.bOpenLockRotate_Cyl_W;
GVL.Q.bOpenLockRotate_Cyl_H:=G_arrCylinder[_i].stOutput.bHome;
GVL.Q.bOpenLockRotate_Cyl_W:=G_arrCylinder[_i].stOutput.bWork;

_i:=E_Cylinder.OpenLockPush2;
//G_arrCylinder[_i].stInput.bHome:=GVL.I.bOpenLockPush2_Cyl_H;
G_arrCylinder[_i].stInput.bHome:=NOT GVL.I.bOpenLockPush2_Cyl_W;
G_arrCylinder[_i].stInput.bWork:=GVL.I.bOpenLockPush2_Cyl_W;
GVL.Q.bOpenLockPush2_Cyl_H:=G_arrCylinder[_i].stOutput.bHome;
GVL.Q.bOpenLockPush2_Cyl_W:=G_arrCylinder[_i].stOutput.bWork;

_i:=E_Cylinder.TakeUcPrevent;
G_arrCylinder[_i].stInput.bWork:=GVL.I.bTakeUcPrevent_Cyl_W;
GVL.Q.bTakeUcPrevent_Cyl_H:=G_arrCylinder[_i].stOutput.bHome;
GVL.Q.bTakeUcPrevent_Cyl_W:=G_arrCylinder[_i].stOutput.bWork;

_i:=E_Cylinder.TakeUcLift;
G_arrCylinder[_i].stInput.bHome:=GVL.I.bTakeUcLift_Cyl_H;
G_arrCylinder[_i].stInput.bWork:=GVL.I.bTakeUcLift_Cyl_W;
GVL.Q.bTakeUcLift_Cyl_H:=G_arrCylinder[_i].stOutput.bHome;
GVL.Q.bTakeUcLift_Cyl_W:=G_arrCylinder[_i].stOutput.bWork;

_i:=E_Cylinder.TakeUcPush;
G_arrCylinder[_i].stInput.bHome:=GVL.I.bTakeUcPush_Cyl_H;
G_arrCylinder[_i].stInput.bWork:=GVL.I.bTakeUcPush_Cyl_W;
GVL.Q.bTakeUcPush_Cyl_H:=G_arrCylinder[_i].stOutput.bHome;
GVL.Q.bTakeUcPush_Cyl_W:=G_arrCylinder[_i].stOutput.bWork;

_i:=E_Cylinder.TakeUcRotate;
G_arrCylinder[_i].stInput.bHome:=GVL.I.bTakeUcRotate_Cyl_H;
G_arrCylinder[_i].stInput.bWork:=GVL.I.bTakeUcRotate_Cyl_W;
GVL.Q.bTakeUcRotate_Cyl_H:=G_arrCylinder[_i].stOutput.bHome;
GVL.Q.bTakeUcRotate_Cyl_W:=G_arrCylinder[_i].stOutput.bWork;

_i:=E_Cylinder.TakeUcStandard;
//G_arrCylinder[_i].stInput.bHome:=GVL.I.bTakeUcStandard_Cyl_H;
//G_arrCylinder[_i].stInput.bWork:=GVL.I.bTakeUcStandard_Cyl_W;
GVL.Q.bTakeUcStandard_Cyl_H:=G_arrCylinder[_i].stOutput.bHome;
GVL.Q.bTakeUcStandard_Cyl_W:=G_arrCylinder[_i].stOutput.bWork;

_i:=E_Cylinder.UnloadFrockPrevent;
G_arrCylinder[_i].stInput.bHome:=GVL.I.bUnloadFrockPrevent_Cyl_H;
G_arrCylinder[_i].stInput.bWork:=GVL.I.bUnloadFrockPrevent_Cyl_W;
GVL.Q.bUnloadFrockPrevent_Cyl_H:=G_arrCylinder[_i].stOutput.bHome;
GVL.Q.bUnloadFrockPrevent_Cyl_W:=G_arrCylinder[_i].stOutput.bWork;

_i:=E_Cylinder.UnloadFrockLift;
G_arrCylinder[_i].stInput.bHome:=GVL.I.bUnloadFrockLift_Cyl_H;
G_arrCylinder[_i].stInput.bWork:=GVL.I.bUnloadFrockLift_Cyl_W;
GVL.Q.bUnloadFrockLift_Cyl_H:=G_arrCylinder[_i].stOutput.bHome;
GVL.Q.bUnloadFrockLift_Cyl_W:=G_arrCylinder[_i].stOutput.bWork;

_i:=E_Cylinder.UnloadFrockPush;
G_arrCylinder[_i].stInput.bHome:=GVL.I.bUnloadFrockPush_Cyl_H;
G_arrCylinder[_i].stInput.bWork:=GVL.I.bUnloadFrockPush_Cyl_W;
GVL.Q.bUnloadFrockPush_Cyl_H:=G_arrCylinder[_i].stOutput.bHome;
GVL.Q.bUnloadFrockPush_Cyl_W:=G_arrCylinder[_i].stOutput.bWork;

_i:=E_Cylinder.TakeUc1Y;
G_arrCylinder[_i].stInput.bHome:=GVL.I.bTakeUc1Y_Cyl_H;
G_arrCylinder[_i].stInput.bWork:=GVL.I.bTakeUc1Y_Cyl_W;
GVL.Q.bTakeUc1Y_Cyl_H:=G_arrCylinder[_i].stOutput.bHome;
GVL.Q.bTakeUc1Y_Cyl_W:=G_arrCylinder[_i].stOutput.bWork;

_i:=E_Cylinder.TakeUc1Z1;
G_arrCylinder[_i].stInput.bHome:=GVL.I.bTakeUc1Z1_Cyl_H;
G_arrCylinder[_i].stInput.bWork:=GVL.I.bTakeUc1Z1_Cyl_W;
GVL.Q.bTakeUc1Z1_Cyl_H:=G_arrCylinder[_i].stOutput.bHome;
GVL.Q.bTakeUc1Z1_Cyl_W:=G_arrCylinder[_i].stOutput.bWork;

_i:=E_Cylinder.TakeUc1Z2;
G_arrCylinder[_i].stInput.bHome:=GVL.I.bTakeUc1Z2_Cyl_H;
G_arrCylinder[_i].stInput.bWork:=GVL.I.bTakeUc1Z2_Cyl_W;
GVL.Q.bTakeUc1Z2_Cyl_H:=G_arrCylinder[_i].stOutput.bHome;
GVL.Q.bTakeUc1Z2_Cyl_W:=G_arrCylinder[_i].stOutput.bWork;

_i:=E_Cylinder.TakeUc1Rotate;
G_arrCylinder[_i].stInput.bHome:=GVL.I.bTakeUc1Rotate_Cyl_H;
G_arrCylinder[_i].stInput.bWork:=GVL.I.bTakeUc1Rotate_Cyl_W;
GVL.Q.bTakeUc1Rotate_Cyl_H:=G_arrCylinder[_i].stOutput.bHome;
GVL.Q.bTakeUc1Rotate_Cyl_W:=G_arrCylinder[_i].stOutput.bWork;

_i:=E_Cylinder.TakeUc1Clamp;
G_arrCylinder[_i].stInput.bHome:=GVL.I.bTakeUc1Clamp_Cyl_H;
//G_arrCylinder[_i].stInput.bWork:=GVL.I.bTakeUc1Clamp_Cyl_W;
GVL.Q.bTakeUc1Clamp_Cyl_H:=G_arrCylinder[_i].stOutput.bHome;
GVL.Q.bTakeUc1Clamp_Cyl_W:=G_arrCylinder[_i].stOutput.bWork;

_i:=E_Cylinder.UnloadUcElevator;
//G_arrCylinder[_i].stInput.bHome:=GVL.I.bUnloadUcElevator_Cyl_H;
//G_arrCylinder[_i].stInput.bWork:=GVL.I.bUnloadUcElevator_Cyl_W;
GVL.Q.bUnloadUcElevator_Cyl_H:=G_arrCylinder[_i].stOutput.bHome;
GVL.Q.bUnloadUcElevator_Cyl_W:=G_arrCylinder[_i].stOutput.bWork;

_i:=E_Cylinder.UnloadUcConveyorPush;
//G_arrCylinder[_i].stInput.bHome:=GVL.I.bUnloadUcConveyorPush_Cyl_H;
//G_arrCylinder[_i].stInput.bWork:=GVL.I.bUnloadUcConveyorPush_Cyl_W;
GVL.Q.bUnloadUcConveyorPush_Cyl_H:=G_arrCylinder[_i].stOutput.bHome;
GVL.Q.bUnloadUcConveyorPush_Cyl_W:=G_arrCylinder[_i].stOutput.bWork;

_i:=E_Cylinder.UnloadFrockConveyorPrevent;
//G_arrCylinder[_i].stInput.bHome:=GVL.I.bUnloadFrockConveyorPrevent_Cyl_H;
//G_arrCylinder[_i].stInput.bWork:=GVL.I.bUnloadFrockConveyorPrevent_Cyl_W;
GVL.Q.bUnloadFrockConveyorPrevent_Cyl_H:=G_arrCylinder[_i].stOutput.bHome;
GVL.Q.bUnloadFrockConveyorPrevent_Cyl_W:=G_arrCylinder[_i].stOutput.bWork;

_i:=E_Cylinder.UnloadFrockConveyorPush;
//G_arrCylinder[_i].stInput.bHome:=GVL.I.bUnloadFrockConveyorPush_Cyl_H;
//G_arrCylinder[_i].stInput.bWork:=GVL.I.bUnloadFrockConveyorPush_Cyl_W;
GVL.Q.bUnloadFrockConveyorPush_Cyl_H:=G_arrCylinder[_i].stOutput.bHome;
GVL.Q.bUnloadFrockConveyorPush_Cyl_W:=G_arrCylinder[_i].stOutput.bWork;

_i:=E_Cylinder.OpenLockElevator;
G_arrCylinder[_i].stInput.bHome:=GVL.I.bOpenLockElevator_Cyl_H;
G_arrCylinder[_i].stInput.bWork:=GVL.I.bOpenLockElevator_Cyl_W;
GVL.Q.bOpenLockElevator_Cyl_H:=G_arrCylinder[_i].stOutput.bHome;
GVL.Q.bOpenLockElevator_Cyl_W:=G_arrCylinder[_i].stOutput.bWork;

_i:=E_Cylinder.OpenLockPin;
G_arrCylinder[_i].stInput.bHome:=GVL.I.bOpenLockPin_Cyl_H;
G_arrCylinder[_i].stInput.bWork:=GVL.I.bOpenLockPin_Cyl_W;
GVL.Q.bOpenLockPin_Cyl_H:=G_arrCylinder[_i].stOutput.bHome;
GVL.Q.bOpenLockPin_Cyl_W:=G_arrCylinder[_i].stOutput.bWork;

_i:=E_Cylinder.TakeUcElevator;
G_arrCylinder[_i].stInput.bHome:=GVL.I.bTakeUcElevator_Cyl_H;
G_arrCylinder[_i].stInput.bWork:=GVL.I.bTakeUcElevator_Cyl_W;
GVL.Q.bTakeUcElevator_Cyl_H:=G_arrCylinder[_i].stOutput.bHome;
GVL.Q.bTakeUcElevator_Cyl_W:=G_arrCylinder[_i].stOutput.bWork;

_i:=E_Cylinder.TakeUcPush1;
G_arrCylinder[_i].stInput.bHome:=GVL.I.bTakeUcPush1_Cyl_H;
G_arrCylinder[_i].stInput.bWork:=GVL.I.bTakeUcPush1_Cyl_W;
GVL.Q.bTakeUcPush1_Cyl_H:=G_arrCylinder[_i].stOutput.bHome;
GVL.Q.bTakeUcPush1_Cyl_W:=G_arrCylinder[_i].stOutput.bWork;

_i:=E_Cylinder.UnloadUcBeltTipper;
G_arrCylinder[_i].stInput.bHome:=GVL.I.bUnloadUcBeltTipper_Cyl_H;
G_arrCylinder[_i].stInput.bWork:=GVL.I.bUnloadUcBeltTipper_Cyl_W;
GVL.Q.bUnloadUcBeltTipper_Cyl_H:=G_arrCylinder[_i].stOutput.bHome;
GVL.Q.bUnloadUcBeltTipper_Cyl_W:=G_arrCylinder[_i].stOutput.bWork;

_i:=E_Cylinder.UnloadUcBeltLift;
G_arrCylinder[_i].stInput.bHome:=GVL.I.bUnloadUcBeltLift_Cyl_H;
G_arrCylinder[_i].stInput.bWork:=GVL.I.bUnloadUcBeltLift_Cyl_W;
GVL.Q.bUnloadUcBeltLift_Cyl_H:=G_arrCylinder[_i].stOutput.bHome;
GVL.Q.bUnloadUcBeltLift_Cyl_W:=G_arrCylinder[_i].stOutput.bWork;

_i:=E_Cylinder.OpenLockTranslation;
G_arrCylinder[_i].stInput.bHome:=GVL.I.bOpenLockTranslation_Cyl_H;
G_arrCylinder[_i].stInput.bWork:=GVL.I.bOpenLockTranslation_Cyl_W;
GVL.Q.bOpenLockTranslation_Cyl_H:=G_arrCylinder[_i].stOutput.bHome;
GVL.Q.bOpenLockTranslation_Cyl_W:=G_arrCylinder[_i].stOutput.bWork;

_i:=E_Cylinder.TakeUcFrockClamp;
G_arrCylinder[_i].stInput.bHome:=GVL.I.bTakeUcFrockClamp_Cyl_H;
G_arrCylinder[_i].stInput.bWork:=GVL.I.bTakeUcFrockClamp_Cyl_W;
GVL.Q.bTakeUcFrockClamp_Cyl_H:=G_arrCylinder[_i].stOutput.bHome;
GVL.Q.bTakeUcFrockClamp_Cyl_W:=G_arrCylinder[_i].stOutput.bWork;
END_ACTION

ACTION A_Info:
_i:=E_Cylinder.Line0Part;
G_arrCylinder[_i].arrInfo[E_Language.Chinese].sName:="主流线分料气缸";
G_arrCylinder[_i].arrInfo[E_Language.English].sName:="Line0Part";
G_arrCylinder[_i].arrInfo[E_Language.Vietnamese].sName:="Xi lanh phân phối dòng chính  ";

_i:=E_Cylinder.Line0Prevent;
G_arrCylinder[_i].arrInfo[E_Language.Chinese].sName:="主流线阻挡气缸";
G_arrCylinder[_i].arrInfo[E_Language.English].sName:="Line0Prevent";
G_arrCylinder[_i].arrInfo[E_Language.Vietnamese].sName:="Dòng chính ngăn chặn các xi lanh  ";

_i:=E_Cylinder.Line0Push;
G_arrCylinder[_i].arrInfo[E_Language.Chinese].sName:="主流线拨料气缸";
G_arrCylinder[_i].arrInfo[E_Language.English].sName:="Line0Push";
G_arrCylinder[_i].arrInfo[E_Language.Vietnamese].sName:="Xi lanh cuộn dòng chính  ";

_i:=E_Cylinder.AcquirePrevent0;
G_arrCylinder[_i].arrInfo[E_Language.Chinese].sName:="接驳线前阻挡气缸";
G_arrCylinder[_i].arrInfo[E_Language.English].sName:="AcquirePrevent0";
G_arrCylinder[_i].arrInfo[E_Language.Vietnamese].sName:="Chặn xi lanh trước dây nối  ";

_i:=E_Cylinder.AcquirePrevent1;
G_arrCylinder[_i].arrInfo[E_Language.Chinese].sName:="接驳线后阻挡气缸";
G_arrCylinder[_i].arrInfo[E_Language.English].sName:="AcquirePrevent1";
G_arrCylinder[_i].arrInfo[E_Language.Vietnamese].sName:="Chặn xi lanh sau khi kết nối  ";

_i:=E_Cylinder.AcquireLift;
G_arrCylinder[_i].arrInfo[E_Language.Chinese].sName:="接驳线顶升气缸";
G_arrCylinder[_i].arrInfo[E_Language.English].sName:="AcquireLift";
G_arrCylinder[_i].arrInfo[E_Language.Vietnamese].sName:="Xi lanh nâng lên dây nối  ";

_i:=E_Cylinder.AcquirePush;
G_arrCylinder[_i].arrInfo[E_Language.Chinese].sName:="接驳模组拨料气缸";
G_arrCylinder[_i].arrInfo[E_Language.English].sName:="AcquirePush";
G_arrCylinder[_i].arrInfo[E_Language.Vietnamese].sName:="Xi lanh kết nối mô-đun  ";

_i:=E_Cylinder.AcquireElevator;
G_arrCylinder[_i].arrInfo[E_Language.Chinese].sName:="接驳模组升降气缸";
G_arrCylinder[_i].arrInfo[E_Language.English].sName:="AcquireElevator";
G_arrCylinder[_i].arrInfo[E_Language.Vietnamese].sName:="Xi lanh nâng mô-đun kết nối  ";

_i:=E_Cylinder.SteeringLift;
G_arrCylinder[_i].arrInfo[E_Language.Chinese].sName:="转向站顶升气缸";
G_arrCylinder[_i].arrInfo[E_Language.English].sName:="SteeringLift";
G_arrCylinder[_i].arrInfo[E_Language.Vietnamese].sName:="Xi lanh hướng về ga nâng lên  ";

_i:=E_Cylinder.SteeringAcquireElevator;
G_arrCylinder[_i].arrInfo[E_Language.Chinese].sName:="转向站接驳升降气缸";
G_arrCylinder[_i].arrInfo[E_Language.English].sName:="SteeringAcquireElevator";
G_arrCylinder[_i].arrInfo[E_Language.Vietnamese].sName:="Trạm lái xe nối với xi lanh nâng  ";

_i:=E_Cylinder.SteeringRotate;
G_arrCylinder[_i].arrInfo[E_Language.Chinese].sName:="转向站旋转气缸";
G_arrCylinder[_i].arrInfo[E_Language.English].sName:="SteeringRotate";
G_arrCylinder[_i].arrInfo[E_Language.Vietnamese].sName:="Quay xi lanh ở trạm rẽ  ";

_i:=E_Cylinder.SteeringAcquireLimit;
G_arrCylinder[_i].arrInfo[E_Language.Chinese].sName:="转向站接驳限位气缸";
G_arrCylinder[_i].arrInfo[E_Language.English].sName:="SteeringAcquireLimit";
G_arrCylinder[_i].arrInfo[E_Language.Vietnamese].sName:="Xi lanh giới hạn kết nối trạm rẽ  ";

_i:=E_Cylinder.OpenLockPrevent;
G_arrCylinder[_i].arrInfo[E_Language.Chinese].sName:="解锁站阻挡气缸";
G_arrCylinder[_i].arrInfo[E_Language.English].sName:="OpenLockPrevent";
G_arrCylinder[_i].arrInfo[E_Language.Vietnamese].sName:="Mở khóa trạm để ngăn chặn xi lanh  ";

_i:=E_Cylinder.OpenLockLift;
G_arrCylinder[_i].arrInfo[E_Language.Chinese].sName:="解锁站顶升气缸";
G_arrCylinder[_i].arrInfo[E_Language.English].sName:="OpenLockLift";
G_arrCylinder[_i].arrInfo[E_Language.Vietnamese].sName:="Mở khóa các xi lanh nâng lên  ";

_i:=E_Cylinder.OpenLockPush;
G_arrCylinder[_i].arrInfo[E_Language.Chinese].sName:="解锁站侧推气缸";
G_arrCylinder[_i].arrInfo[E_Language.English].sName:="OpenLockPush";
G_arrCylinder[_i].arrInfo[E_Language.Vietnamese].sName:="Mở khóa xi lanh đẩy ga  ";

_i:=E_Cylinder.OpenLockRotate;
G_arrCylinder[_i].arrInfo[E_Language.Chinese].sName:="解锁站旋转气缸";
G_arrCylinder[_i].arrInfo[E_Language.English].sName:="OpenLockRotate";
G_arrCylinder[_i].arrInfo[E_Language.Vietnamese].sName:="Mở khóa trạm quay xi lanh  ";

_i:=E_Cylinder.OpenLockPush2;
G_arrCylinder[_i].arrInfo[E_Language.Chinese].sName:="解锁站侧推气缸2";
G_arrCylinder[_i].arrInfo[E_Language.English].sName:="OpenLockPush2";
G_arrCylinder[_i].arrInfo[E_Language.Vietnamese].sName:="Mở khóa ga đẩy xi lanh 2  ";

_i:=E_Cylinder.TakeUcPrevent;
G_arrCylinder[_i].arrInfo[E_Language.Chinese].sName:="取UC站阻挡气缸";
G_arrCylinder[_i].arrInfo[E_Language.English].sName:="TakeUcPrevent";
G_arrCylinder[_i].arrInfo[E_Language.Vietnamese].sName:="Lấy trụ UC để ngăn chặn xi lanh  ";

_i:=E_Cylinder.TakeUcLift;
G_arrCylinder[_i].arrInfo[E_Language.Chinese].sName:="取UC站顶升气缸";
G_arrCylinder[_i].arrInfo[E_Language.English].sName:="TakeUcLift";
G_arrCylinder[_i].arrInfo[E_Language.Vietnamese].sName:="Lấy xi lanh nâng lên từ trạm UC  ";

_i:=E_Cylinder.TakeUcPush;
G_arrCylinder[_i].arrInfo[E_Language.Chinese].sName:="取UC站侧推气缸";
G_arrCylinder[_i].arrInfo[E_Language.English].sName:="TakeUcPush";
G_arrCylinder[_i].arrInfo[E_Language.Vietnamese].sName:="Lấy ống đẩy bên ga UC  ";

_i:=E_Cylinder.TakeUcRotate;
G_arrCylinder[_i].arrInfo[E_Language.Chinese].sName:="取UC站旋转气缸";
G_arrCylinder[_i].arrInfo[E_Language.English].sName:="TakeUcRotate";
G_arrCylinder[_i].arrInfo[E_Language.Vietnamese].sName:="Lấy xi lanh quay từ trạm UC  ";

_i:=E_Cylinder.TakeUcStandard;
G_arrCylinder[_i].arrInfo[E_Language.Chinese].sName:="取UC站校平气缸";
G_arrCylinder[_i].arrInfo[E_Language.English].sName:="TakeUcStandard";
G_arrCylinder[_i].arrInfo[E_Language.Vietnamese].sName:="Lấy xi lanh bằng phẳng từ trạm UC  ";

_i:=E_Cylinder.UnloadFrockPrevent;
G_arrCylinder[_i].arrInfo[E_Language.Chinese].sName:="下工装站阻挡气缸";
G_arrCylinder[_i].arrInfo[E_Language.English].sName:="UnloadFrockPrevent";
G_arrCylinder[_i].arrInfo[E_Language.Vietnamese].sName:="Trạm dừng xi lanh  ";

_i:=E_Cylinder.UnloadFrockLift;
G_arrCylinder[_i].arrInfo[E_Language.Chinese].sName:="下工装站顶升气缸";
G_arrCylinder[_i].arrInfo[E_Language.English].sName:="UnloadFrockLift";
G_arrCylinder[_i].arrInfo[E_Language.Vietnamese].sName:="Xi lanh nâng lên xuống ga  ";

_i:=E_Cylinder.UnloadFrockPush;
G_arrCylinder[_i].arrInfo[E_Language.Chinese].sName:="下工装站拨料气缸";
G_arrCylinder[_i].arrInfo[E_Language.English].sName:="UnloadFrockPush";
G_arrCylinder[_i].arrInfo[E_Language.Vietnamese].sName:="Xi lanh vật liệu trạm tiếp theo  ";

_i:=E_Cylinder.TakeUc1Y;
G_arrCylinder[_i].arrInfo[E_Language.Chinese].sName:="取UC模组平移Y气缸";
G_arrCylinder[_i].arrInfo[E_Language.English].sName:="TakeUc1Y";
G_arrCylinder[_i].arrInfo[E_Language.Vietnamese].sName:="Lấy mô-đun UC và chuyển xi lanh Y  ";

_i:=E_Cylinder.TakeUc1Z1;
G_arrCylinder[_i].arrInfo[E_Language.Chinese].sName:="取UC模组升降Z1气缸";
G_arrCylinder[_i].arrInfo[E_Language.English].sName:="TakeUc1Z1";
G_arrCylinder[_i].arrInfo[E_Language.Vietnamese].sName:="Nâng xi lanh Z1 bằng mô-đun UC  ";

_i:=E_Cylinder.TakeUc1Z2;
G_arrCylinder[_i].arrInfo[E_Language.Chinese].sName:="取UC模组升降Z2气缸";
G_arrCylinder[_i].arrInfo[E_Language.English].sName:="TakeUc1Z2";
G_arrCylinder[_i].arrInfo[E_Language.Vietnamese].sName:="Lấy mô-đun UC nâng xi lanh Z2  ";

_i:=E_Cylinder.TakeUc1Rotate;
G_arrCylinder[_i].arrInfo[E_Language.Chinese].sName:="取UC模组旋转气缸";
G_arrCylinder[_i].arrInfo[E_Language.English].sName:="TakeUc1Rotate";
G_arrCylinder[_i].arrInfo[E_Language.Vietnamese].sName:="Lấy xi lanh quay trong mô-đun UC  ";

_i:=E_Cylinder.TakeUc1Clamp;
G_arrCylinder[_i].arrInfo[E_Language.Chinese].sName:="取UC模组夹紧气缸";
G_arrCylinder[_i].arrInfo[E_Language.English].sName:="TakeUc1Clamp";
G_arrCylinder[_i].arrInfo[E_Language.Vietnamese].sName:="Lấy mô-đun UC kẹp xi lanh  ";

_i:=E_Cylinder.UnloadUcElevator;
G_arrCylinder[_i].arrInfo[E_Language.Chinese].sName:="下UC皮带升降气缸";
G_arrCylinder[_i].arrInfo[E_Language.English].sName:="UnloadUcElevator";
G_arrCylinder[_i].arrInfo[E_Language.Vietnamese].sName:="Ống nâng dưới vành đai UC  ";

_i:=E_Cylinder.UnloadUcConveyorPush;
G_arrCylinder[_i].arrInfo[E_Language.Chinese].sName:="下UC皮带拨料气缸";
G_arrCylinder[_i].arrInfo[E_Language.English].sName:="UnloadUcConveyorPush";
G_arrCylinder[_i].arrInfo[E_Language.Vietnamese].sName:="Xi lanh dưới vành đai UC  ";

_i:=E_Cylinder.UnloadFrockConveyorPrevent;
G_arrCylinder[_i].arrInfo[E_Language.Chinese].sName:="下工装皮带升降气缸";
G_arrCylinder[_i].arrInfo[E_Language.English].sName:="UnloadFrockConveyorPrevent";
G_arrCylinder[_i].arrInfo[E_Language.Vietnamese].sName:="Dây chuyền nâng xi lanh  ";

_i:=E_Cylinder.UnloadFrockConveyorPush;
G_arrCylinder[_i].arrInfo[E_Language.Chinese].sName:="下工装皮带拨料气缸";
G_arrCylinder[_i].arrInfo[E_Language.English].sName:="UnloadFrockConveyorPush";
G_arrCylinder[_i].arrInfo[E_Language.Vietnamese].sName:="Xi lanh dây buộc công nhân  ";

_i:=E_Cylinder.OpenLockElevator;
G_arrCylinder[_i].arrInfo[E_Language.Chinese].sName:="解锁站升降气缸";
G_arrCylinder[_i].arrInfo[E_Language.English].sName:="OpenLockElevator";
G_arrCylinder[_i].arrInfo[E_Language.Vietnamese].sName:="Mở khóa trạm nâng xi lanh  ";

_i:=E_Cylinder.OpenLockPin;
G_arrCylinder[_i].arrInfo[E_Language.Chinese].sName:="解锁站按压气缸";
G_arrCylinder[_i].arrInfo[E_Language.English].sName:="OpenLockPin";
G_arrCylinder[_i].arrInfo[E_Language.Vietnamese].sName:="Mở khóa trạm nhấn xi lanh  ";

_i:=E_Cylinder.TakeUcElevator;
G_arrCylinder[_i].arrInfo[E_Language.Chinese].sName:="取UC站升降气缸";
G_arrCylinder[_i].arrInfo[E_Language.English].sName:="TakeUcElevator";
G_arrCylinder[_i].arrInfo[E_Language.Vietnamese].sName:="Lấy xi lanh nâng từ trạm UC  ";

_i:=E_Cylinder.TakeUcPush1;
G_arrCylinder[_i].arrInfo[E_Language.Chinese].sName:="取UC站侧推气缸1";
G_arrCylinder[_i].arrInfo[E_Language.English].sName:="TakeUcPush1";
G_arrCylinder[_i].arrInfo[E_Language.Vietnamese].sName:="Lấy xi lanh 1 đẩy bên ga UC  ";

_i:=E_Cylinder.UnloadUcBeltTipper;
G_arrCylinder[_i].arrInfo[E_Language.Chinese].sName:="下UC皮带翻转气缸";
G_arrCylinder[_i].arrInfo[E_Language.English].sName:="UnloadUcBeltTipper";
G_arrCylinder[_i].arrInfo[E_Language.Vietnamese].sName:="Phía dưới vành đai xoay xi lanh  ";

_i:=E_Cylinder.UnloadUcBeltLift;
G_arrCylinder[_i].arrInfo[E_Language.Chinese].sName:="下UC皮带顶升气缸";
G_arrCylinder[_i].arrInfo[E_Language.English].sName:="UnloadUcBeltLift";
G_arrCylinder[_i].arrInfo[E_Language.Vietnamese].sName:="Xi lanh nâng lên phía dưới vành đai UC  ";

_i:=E_Cylinder.OpenLockTranslation;
G_arrCylinder[_i].arrInfo[E_Language.Chinese].sName:="解锁站解锁平移气缸";
G_arrCylinder[_i].arrInfo[E_Language.English].sName:="OpenLockTranslation";
G_arrCylinder[_i].arrInfo[E_Language.Vietnamese].sName:="Trạm mở khóa mở xi lanh dịch chuyển  ";

_i:=E_Cylinder.TakeUcFrockClamp;
G_arrCylinder[_i].arrInfo[E_Language.Chinese].sName:="取UC站工装夹紧气缸";
G_arrCylinder[_i].arrInfo[E_Language.English].sName:="TakeUcFrockClamp";
G_arrCylinder[_i].arrInfo[E_Language.Vietnamese].sName:="Lấy xi lanh bị kẹp ở trạm UC";

_i:=E_Cylinder.OpenLockPressPush;
G_arrCylinder[_i].arrInfo[E_Language.Chinese].sName:="解锁站解压侧推气缸";
G_arrCylinder[_i].arrInfo[E_Language.English].sName:="OpenLockPressPush";
G_arrCylinder[_i].arrInfo[E_Language.Vietnamese].sName:="OpenLockPressPush";

_i:=E_Cylinder.OpenLockPressRotate;
G_arrCylinder[_i].arrInfo[E_Language.Chinese].sName:="解锁站解压旋转气缸";
G_arrCylinder[_i].arrInfo[E_Language.English].sName:="OpenLockPressRotate";
G_arrCylinder[_i].arrInfo[E_Language.Vietnamese].sName:="OpenLockPressRotate";

_i:=E_Cylinder.AcquirePrevent2;
G_arrCylinder[_i].arrInfo[E_Language.Chinese].sName:="接驳线前前阻挡气缸";
G_arrCylinder[_i].arrInfo[E_Language.English].sName:="AcquirePrevent2";
G_arrCylinder[_i].arrInfo[E_Language.Vietnamese].sName:="AcquirePrevent2";

_i:=E_Cylinder.Line0PushElevator;
G_arrCylinder[_i].arrInfo[E_Language.Chinese].sName:="主流线拨料升降气缸";
G_arrCylinder[_i].arrInfo[E_Language.English].sName:="Line0PushElevator";
G_arrCylinder[_i].arrInfo[E_Language.Vietnamese].sName:="Line0PushElevator";
END_ACTION

ACTION A_InOut:
//输出信号
//结构体->Bool数组1->加延迟->Bool数组2->字节数组
//输入信号
//字节数组->Bool数组->加延迟->Bool数组2->结构体




FOR _i:=0 TO 7 BY 1 DO
	FOR _t:=0 TO 15 BY 1 DO
		IF GVL.stSetting.bDryRun AND _i=6 THEN
			_fbPulse(PT:=T#1S , Q=> _arrInput[_i,_t]);
		ELSE
			_arrTonInput[_i,_t](IN:=GVL_IO.I_Temp[_i,_t] , PT:=TO_TIME(GVL_Data.stRecipe.arrInputTon[_i,_t]) , Q=>_arrInput[_i,_t] , ET=> );
		END_IF
	END_FOR
END_FOR

FOR _i:=0 TO 6 BY 1 DO
	FOR _t:=0 TO 15 BY 1 DO
		IF NOT G_stSystem.stMode.bSetting THEN
			_arrTonOutput[_i,_t](IN:=_arrOutput[_i,_t] , PT:=TO_TIME(GVL_Data.stRecipe.arrOutputTon[_i,_t]) , Q=>GVL_IO.Q_Temp[_i,_t] , ET=> );
		END_IF
	END_FOR
END_FOR


Data_TO_Data(ADR(_arrInput),SIZEOF(_arrInput),ADR(GVL.I),SIZEOF(GVL.I));
Data_TO_Data(ADR(GVL.Q),SIZEOF(GVL.Q),ADR(_arrOutput),SIZEOF(_arrOutput));


ArrayBool_TO_ArrayByte(ADR(GVL_IO.Q_Temp),SIZEOF(GVL_IO.Q_Temp),ADR(GVL_IO.Q),SIZEOF(GVL_IO.Q));
ArrayByte_TO_ArrayBool(ADR(GVL_IO.I),SIZEOF(GVL_IO.I),ADR(GVL_IO.I_Temp),SIZEOF(GVL_IO.I_Temp));




// IO屏蔽
IF GVL_Data.stRecipe.eMachineType<>_eMachineType THEN
	_boolTemp:=ADR(GVL.stShield_I);
	FOR _i:=0 TO SIZEOF(GVL.stShield_I)-1 BY 1 DO
		_boolTemp[_i]:=FALSE;
	END_FOR
	_boolTemp:=ADR(GVL.stShield_Q);
	FOR _i:=0 TO SIZEOF(GVL.stShield_Q)-1 BY 1 DO
		_boolTemp[_i]:=FALSE;
	END_FOR
	_eMachineType:=GVL_Data.stRecipe.eMachineType;
END_IF



CASE GVL_Data.stRecipe.eMachineType OF
	E_MachineType._200:
		GVL.stShield_I[0,5]:=TRUE;		
		GVL.stShield_I[0,6]:=TRUE;		
		GVL.stShield_I[0,7]:=TRUE;		
		GVL.stShield_I[0,8]:=TRUE;		
		GVL.stShield_I[0,9]:=TRUE;		
		GVL.stShield_I[0,10]:=TRUE;		
		GVL.stShield_I[0,11]:=TRUE;		
		GVL.stShield_I[0,12]:=TRUE;	
		GVL.stShield_I[3,10]:=TRUE;
		GVL.stShield_I[3,11]:=TRUE;
		GVL.stShield_I[3,12]:=TRUE;
		GVL.stShield_I[3,13]:=TRUE;
		GVL.stShield_I[6,14]:=TRUE;
		
		GVL.stShield_Q[0,7]:=TRUE;
		GVL.stShield_Q[0,12]:=TRUE;
		GVL.stShield_Q[0,13]:=TRUE;
		GVL.stShield_Q[3,10]:=TRUE;
		GVL.stShield_Q[3,11]:=TRUE;
		GVL.stShield_Q[3,12]:=TRUE;
		GVL.stShield_Q[3,13]:=TRUE;
		GVL.stShield_Q[5,11]:=TRUE;
		
		FOR _i:=0 TO 15 BY 1 DO
			GVL.stShield_I[7,_i]:=TRUE;
			GVL.stShield_Q[6,_i]:=TRUE;
		END_FOR
	E_MachineType._367:
		FOR _i:=6 TO 15 BY 1 DO
			GVL.stShield_I[1,_i]:=TRUE;
			GVL.stShield_Q[1,_i]:=TRUE;
		END_FOR
	
		GVL.stShield_I[0,5]:=TRUE;		
		GVL.stShield_I[0,6]:=FALSE;		
		GVL.stShield_I[0,7]:=TRUE;				
		GVL.stShield_I[0,10]:=TRUE;		
		GVL.stShield_I[0,11]:=TRUE;		
		GVL.stShield_I[0,12]:=FALSE;	
		GVL.stShield_I[0,13]:=TRUE;
		GVL.stShield_I[0,14]:=TRUE;
		GVL.stShield_I[0,15]:=TRUE;
		GVL.stShield_I[3,14]:=TRUE;
		GVL.stShield_I[3,15]:=TRUE;
		GVL.stShield_I[4,0]:=TRUE;
		GVL.stShield_I[4,1]:=TRUE;
		GVL.stShield_I[6,3]:=TRUE;
		GVL.stShield_I[6,4]:=TRUE;
		GVL.stShield_I[5,6]:=TRUE;
		GVL.stShield_I[5,7]:=TRUE;
		GVL.stShield_I[5,8]:=TRUE;
		GVL.stShield_I[5,9]:=TRUE;
		GVL.stShield_I[5,10]:=TRUE;
		GVL.stShield_I[5,11]:=TRUE;
		GVL.stShield_I[5,12]:=TRUE;
		GVL.stShield_I[5,13]:=TRUE;
		GVL.stShield_I[5,14]:=TRUE;
		GVL.stShield_I[5,15]:=TRUE;
		GVL.stShield_I[6,13]:=TRUE;
		GVL.stShield_I[6,14]:=TRUE;
		
		GVL.stShield_Q[0,7]:=TRUE;
		GVL.stShield_Q[0,14]:=TRUE;
		GVL.stShield_Q[0,15]:=TRUE;
		GVL.stShield_Q[3,14]:=TRUE;
		GVL.stShield_Q[3,15]:=TRUE;
		GVL.stShield_Q[4,0]:=TRUE;
		GVL.stShield_Q[4,1]:=TRUE;
		GVL.stShield_Q[5,6]:=TRUE;
		GVL.stShield_Q[5,7]:=TRUE;
		GVL.stShield_Q[5,11]:=TRUE;
		GVL.stShield_Q[5,12]:=TRUE;
		GVL.stShield_Q[5,13]:=TRUE;
		GVL.stShield_Q[5,14]:=TRUE;
		GVL.stShield_Q[5,15]:=TRUE;
		
		FOR _i:=0 TO 15 BY 1 DO
			GVL.stShield_I[7,_i]:=TRUE;
			GVL.stShield_Q[6,_i]:=TRUE;
		END_FOR
	E_MachineType._373:
		GVL.stShield_I[0,5]:=TRUE;		
		GVL.stShield_I[0,6]:=TRUE;		
		GVL.stShield_I[0,7]:=TRUE;		
		GVL.stShield_I[0,8]:=TRUE;		
		GVL.stShield_I[0,9]:=TRUE;		
		GVL.stShield_I[0,10]:=TRUE;		
		GVL.stShield_I[0,11]:=TRUE;		
		GVL.stShield_I[0,12]:=TRUE;	
		GVL.stShield_I[0,13]:=FALSE;	
		GVL.stShield_I[0,14]:=FALSE;	
		GVL.stShield_I[0,15]:=FALSE;	
		GVL.stShield_I[2,0]:=TRUE;
		GVL.stShield_I[2,1]:=TRUE;
		GVL.stShield_I[2,4]:=TRUE;
		GVL.stShield_I[2,5]:=TRUE;
		GVL.stShield_I[3,0]:=TRUE;
		GVL.stShield_I[3,1]:=TRUE;
		GVL.stShield_I[3,10]:=TRUE;
		GVL.stShield_I[3,11]:=TRUE;
		GVL.stShield_I[3,12]:=TRUE;
		GVL.stShield_I[3,13]:=TRUE;
		GVL.stShield_I[3,14]:=TRUE;
		GVL.stShield_I[3,15]:=TRUE;
		GVL.stShield_I[4,0]:=TRUE;
		GVL.stShield_I[4,1]:=TRUE;
		GVL.stShield_I[4,8]:=TRUE;
		GVL.stShield_I[4,9]:=TRUE;
		GVL.stShield_I[5,10]:=TRUE;
		GVL.stShield_I[5,11]:=TRUE;
		GVL.stShield_I[5,12]:=TRUE;
		GVL.stShield_I[5,13]:=TRUE;
		GVL.stShield_I[5,14]:=TRUE;
		GVL.stShield_I[5,15]:=TRUE;
		GVL.stShield_I[6,13]:=TRUE;
		GVL.stShield_I[6,14]:=FALSE;
		
		GVL.stShield_Q[0,7]:=TRUE;
		GVL.stShield_Q[0,12]:=TRUE;		
		GVL.stShield_Q[0,13]:=TRUE;
		GVL.stShield_Q[2,0]:=TRUE;
		GVL.stShield_Q[2,1]:=TRUE;
		GVL.stShield_Q[2,4]:=TRUE;
		GVL.stShield_Q[2,5]:=TRUE;				
		GVL.stShield_Q[3,0]:=TRUE;
		GVL.stShield_Q[3,1]:=TRUE;
		GVL.stShield_Q[3,10]:=TRUE;
		GVL.stShield_Q[3,11]:=TRUE;
		GVL.stShield_Q[3,12]:=TRUE;
		GVL.stShield_Q[3,13]:=TRUE;
		GVL.stShield_Q[3,14]:=TRUE;
		GVL.stShield_Q[3,15]:=TRUE;
		GVL.stShield_Q[4,0]:=TRUE;
		GVL.stShield_Q[4,1]:=TRUE;
		GVL.stShield_Q[4,8]:=TRUE;
		GVL.stShield_Q[4,9]:=TRUE;
		GVL.stShield_Q[5,11]:=TRUE;
		GVL.stShield_Q[5,12]:=TRUE;
		GVL.stShield_Q[5,13]:=TRUE;
		GVL.stShield_Q[5,14]:=TRUE;
		GVL.stShield_Q[5,15]:=TRUE;
		
		FOR _i:=0 TO 15 BY 1 DO
			GVL.stShield_I[7,_i]:=TRUE;
			GVL.stShield_Q[6,_i]:=TRUE;
		END_FOR
	E_MachineType._069:
		GVL.stShield_I[0,5]:=TRUE;		
		GVL.stShield_I[0,6]:=TRUE;		
		GVL.stShield_I[0,7]:=TRUE;		
		GVL.stShield_I[0,8]:=TRUE;		
		GVL.stShield_I[0,9]:=TRUE;		
		GVL.stShield_I[0,10]:=TRUE;		
		GVL.stShield_I[0,11]:=TRUE;		
		GVL.stShield_I[0,12]:=TRUE;	
		GVL.stShield_I[2,0]:=TRUE;
		GVL.stShield_I[2,1]:=TRUE;
		GVL.stShield_I[2,4]:=TRUE;
		GVL.stShield_I[2,5]:=TRUE;
		GVL.stShield_I[3,10]:=TRUE;
		GVL.stShield_I[3,11]:=TRUE;
		GVL.stShield_I[3,12]:=TRUE;
		GVL.stShield_I[3,13]:=TRUE;
		GVL.stShield_I[3,14]:=TRUE;
		GVL.stShield_I[3,15]:=TRUE;
		GVL.stShield_I[4,0]:=TRUE;
		GVL.stShield_I[4,1]:=TRUE;
		GVL.stShield_I[5,6]:=TRUE;
		GVL.stShield_I[5,7]:=TRUE;
		GVL.stShield_I[5,8]:=TRUE;
		GVL.stShield_I[5,9]:=TRUE;
		GVL.stShield_I[5,10]:=TRUE;
		GVL.stShield_I[5,11]:=TRUE;
		GVL.stShield_I[5,12]:=TRUE;
		GVL.stShield_I[5,13]:=TRUE;
		GVL.stShield_I[5,14]:=TRUE;
		GVL.stShield_I[5,15]:=TRUE;
		GVL.stShield_I[6,13]:=TRUE;
		GVL.stShield_I[6,14]:=TRUE;
		
		GVL.stShield_Q[0,7]:=TRUE;
		GVL.stShield_Q[0,12]:=TRUE;
		GVL.stShield_Q[0,13]:=TRUE;
		GVL.stShield_Q[2,0]:=TRUE;
		GVL.stShield_Q[2,1]:=TRUE;
		GVL.stShield_Q[2,4]:=TRUE;
		GVL.stShield_Q[2,5]:=TRUE;
		GVL.stShield_Q[3,10]:=TRUE;
		GVL.stShield_Q[3,11]:=TRUE;
		GVL.stShield_Q[3,12]:=TRUE;
		GVL.stShield_Q[3,13]:=TRUE;
		GVL.stShield_Q[3,14]:=TRUE;
		GVL.stShield_Q[3,15]:=TRUE;
		GVL.stShield_Q[4,0]:=TRUE;
		GVL.stShield_Q[4,1]:=TRUE;
		GVL.stShield_Q[5,11]:=TRUE;
		GVL.stShield_Q[5,12]:=TRUE;
		GVL.stShield_Q[5,13]:=TRUE;
		GVL.stShield_Q[5,14]:=TRUE;
		GVL.stShield_Q[5,15]:=TRUE;
	
		FOR _i:=0 TO 15 BY 1 DO
			GVL.stShield_I[7,_i]:=TRUE;
			GVL.stShield_Q[6,_i]:=TRUE;
		END_FOR
	E_MachineType._311:
		GVL.stShield_I[0,5]:=FALSE;		
		GVL.stShield_I[0,6]:=TRUE;		
		GVL.stShield_I[0,7]:=TRUE;		
		GVL.stShield_I[0,8]:=TRUE;		
		GVL.stShield_I[0,9]:=TRUE;		
		GVL.stShield_I[0,10]:=TRUE;		
		GVL.stShield_I[0,11]:=TRUE;		
		GVL.stShield_I[0,12]:=TRUE;
		GVL.stShield_I[2,0]:=TRUE;
		GVL.stShield_I[2,1]:=TRUE;
		GVL.stShield_I[2,4]:=TRUE;
		GVL.stShield_I[2,5]:=TRUE;	
		GVL.stShield_I[3,0]:=TRUE;
		GVL.stShield_I[3,1]:=TRUE;
		GVL.stShield_I[3,10]:=TRUE;
		GVL.stShield_I[3,11]:=TRUE;
		GVL.stShield_I[3,12]:=TRUE;
		GVL.stShield_I[3,13]:=TRUE;
		GVL.stShield_I[3,14]:=TRUE;
		GVL.stShield_I[3,15]:=TRUE;
		GVL.stShield_I[4,0]:=TRUE;
		GVL.stShield_I[4,1]:=TRUE;
		GVL.stShield_I[5,6]:=TRUE;
		GVL.stShield_I[5,7]:=TRUE;
		GVL.stShield_I[5,8]:=TRUE;
		GVL.stShield_I[5,9]:=TRUE;
		GVL.stShield_I[5,10]:=TRUE;
		GVL.stShield_I[5,11]:=TRUE;
		GVL.stShield_I[5,12]:=TRUE;
		GVL.stShield_I[5,13]:=TRUE;
		GVL.stShield_I[5,14]:=TRUE;
		GVL.stShield_I[5,15]:=TRUE;
		GVL.stShield_I[6,13]:=TRUE;
		GVL.stShield_I[6,14]:=TRUE;
		
		GVL.stShield_Q[0,7]:=TRUE;
		GVL.stShield_Q[0,12]:=TRUE;
		GVL.stShield_Q[0,13]:=TRUE;
		GVL.stShield_Q[2,0]:=TRUE;
		GVL.stShield_Q[2,1]:=TRUE;
		GVL.stShield_Q[2,4]:=TRUE;
		GVL.stShield_Q[2,5]:=TRUE;
		GVL.stShield_Q[3,0]:=TRUE;
		GVL.stShield_Q[3,1]:=TRUE;
		GVL.stShield_Q[3,10]:=TRUE;
		GVL.stShield_Q[3,11]:=TRUE;
		GVL.stShield_Q[3,12]:=TRUE;
		GVL.stShield_Q[3,13]:=TRUE;
		GVL.stShield_Q[3,14]:=TRUE;
		GVL.stShield_Q[3,15]:=TRUE;
		GVL.stShield_Q[4,0]:=TRUE;
		GVL.stShield_Q[4,1]:=TRUE;
		GVL.stShield_Q[5,11]:=TRUE;
		GVL.stShield_Q[5,12]:=TRUE;
		GVL.stShield_Q[5,13]:=TRUE;
		GVL.stShield_Q[5,14]:=TRUE;
		GVL.stShield_Q[5,15]:=TRUE;
END_CASE
END_ACTION

ACTION A_Line:
GVL.arrFbLine[E_LineAxis.Acquire](System:=G_stSystem , Moving=>GVL.Q.bAcquireAxis );
GVL.arrFbLine[E_LineAxis.UnloadForck](System:=G_stSystem , Moving=>GVL.Q.bUnloadFrock );
GVL.arrFbLine[E_LineAxis.UnloadUc](System:=G_stSystem , Moving=>GVL.Q.bUnloadUcAxis );
GVL.arrFbLine[E_LineAxis.Dismantling](System:=G_stSystem , Moving=>GVL.Q.bDismantlingAxis );
GVL.arrFbLine[E_LineAxis.AcquireFront](System:=G_stSystem , Moving=>GVL.Q.bAcquireFrontAxis );

IF G_stSystem.stMode.bAutoRunning THEN
	GVL.arrFbLine[E_LineAxis.Acquire].M_Jog(1);
	GVL.arrFbLine[E_LineAxis.UnloadForck].M_Jog(1);
	GVL.arrFbLine[E_LineAxis.Dismantling].M_Jog(1);
	GVL.arrFbLine[E_LineAxis.AcquireFront].M_Jog(1);
END_IF
END_ACTION

END_PROGRAM

// ---- POUs/Device/ArrayBool_TO_ArrayByte.TcPOU
FUNCTION ArrayBool_TO_ArrayByte 
VAR_INPUT
	In:					POINTER TO BOOL;// Bool数组
	InLen:				INT;// sizeof(In)
	Out:				POINTER TO BYTE;// Byte数组
	OutLen:				INT;// sizeof(Out)
END_VAR
VAR
	i:					INT;
	t:					INT;
	temp:				ARRAY[0..7] OF BOOL;
	inCount:			INT;
END_VAR

IF InLen<>OutLen*8 THEN
	RETURN;
END_IF

FOR i:=0 TO OutLen-1 BY 1 DO
	FOR t:=0 TO 7 BY 1 DO
		temp[t]:=In[inCount];
		inCount:=inCount+1;
	END_FOR
	Out[i]:=ArrayBool_TO_Byte(ADR(temp),SIZEOF(temp));
END_FOR

END_FUNCTION

// ---- POUs/Device/ArrayBool_TO_Byte.TcPOU
FUNCTION ArrayBool_TO_Byte : BYTE
VAR_INPUT
	In:				POINTER TO	BOOL;
	InLen:			INT;// sizeof(In)
END_VAR
VAR
END_VAR

IF InLen<>8 THEN
	RETURN;
END_IF

ArrayBool_TO_Byte.0:=In[0];
ArrayBool_TO_Byte.1:=In[1];
ArrayBool_TO_Byte.2:=In[2];
ArrayBool_TO_Byte.3:=In[3];
ArrayBool_TO_Byte.4:=In[4];
ArrayBool_TO_Byte.5:=In[5];
ArrayBool_TO_Byte.6:=In[6];
ArrayBool_TO_Byte.7:=In[7];

END_FUNCTION

// ---- POUs/Device/ArrayByte_TO_ArrayBool.TcPOU
FUNCTION ArrayByte_TO_ArrayBool 
VAR_INPUT
	In:					POINTER TO BYTE;// Byte数组
	InLen:				INT;// Sizeof(In)
	Out:				POINTER TO BOOL;// Bool数组
	OutLen:				INT;// sizeof(Out)
END_VAR
VAR
	i:					INT;
	t:					INT;
	outCount:			INT;
	temp:				ARRAY[0..7] OF BOOL;
END_VAR

FOR i:=0 TO InLen-1 BY 1 DO
	temp:=Byte_TO_ArrayBool(ADR(In[i]));
	FOR t:=0 TO 7 BY 1 DO
		IF outCount<OutLen THEN
			Out[outCount]:=temp[t];
			outCount:=outCount+1;
		END_IF
	END_FOR
END_FOR

END_FUNCTION

// ---- POUs/Device/Byte_TO_ArrayBool.TcPOU
FUNCTION Byte_TO_ArrayBool :ARRAY[0..7] OF BOOL;
VAR_INPUT
	In:				POINTER TO	BYTE;
END_VAR
VAR
END_VAR

Byte_TO_ArrayBool[0]:=In^.0;
Byte_TO_ArrayBool[1]:=In^.1;
Byte_TO_ArrayBool[2]:=In^.2;
Byte_TO_ArrayBool[3]:=In^.3;
Byte_TO_ArrayBool[4]:=In^.4;
Byte_TO_ArrayBool[5]:=In^.5;
Byte_TO_ArrayBool[6]:=In^.6;
Byte_TO_ArrayBool[7]:=In^.7;

END_FUNCTION

// ---- POUs/P_StationAcquire.TcPOU
PROGRAM P_StationAcquire
VAR
	_station:					REFERENCE TO ST_SystemStation;
	_bEnable:					BOOL;
	_eLoadClose:				E_LoadClose;// 关闭状态缓存
	_eLoadClass:				E_LoadClass;// 优先级缓存
END_VAR

_station REF= G_arrStation[E_Station.Acquire];
_station.arrName[E_Language.Chinese]:="接驳站";
_station.arrName[E_Language.Vietnamese]:="Trạm truy cập";
_bEnable:=NOT GVL.stSetting.arrStationShield[E_Station.Acquire] AND E_MachineType._367 <> GVL_Data.stRecipe.eMachineType;
 GVL.stSetting.arrStationShield[E_Station.Acquire]:=GVL.stSetting.bManualLoad;


A_Auto();
A_Home();

GVL._arrAutoTimer[E_Timer.Line0PriorityOnDelay](IN:=GVL.I.bLine0Check1, PT:=TO_TIME(GVL_Data.stRecipe.arrAutoTon[E_Timer.Line0PriorityOnDelay]), Q=>GVL._arrAutoTimerOut[E_Timer.Line0PriorityOnDelay] , ET=> );
GVL._arrAutoTimer[E_Timer.Line0PriorityOffDelay](IN:=NOT GVL.I.bLine0Check1 AND NOT GVL.I.bLine0Check2, PT:=TO_TIME(GVL_Data.stRecipe.arrAutoTon[E_Timer.Line0PriorityOffDelay]), Q=>GVL._arrAutoTimerOut[E_Timer.Line0PriorityOffDelay] , ET=> );

IF GVL._arrAutoTimerOut[E_Timer.Line0PriorityOnDelay] THEN
	GVL.stSetting.bLine0Priority:=TRUE;
ELSIF GVL._arrAutoTimerOut[E_Timer.Line0PriorityOffDelay] THEN
	GVL.stSetting.bLine0Priority:=FALSE;	
END_IF

ACTION A_Auto:
CASE _station.iStepNow OF
	1000:
		_station.arrInfo[E_Language.Chinese]:="初始化完成等待启动";
		IF _bEnable  THEN
			_station.iStepNext:=1100;
		END_IF
	1100:
		_station.arrInfo[E_Language.Chinese]:="缓存状态";
		_eLoadClass:=GVL_Data.stRecipe.eLoadClass;
		_eLoadClose:=GVL_Data.stRecipe.eLoadClose;
		_station.iStepNext:=1200;	
	1200:
		_station.arrInfo[E_Language.Chinese]:="请求上料";
		CASE _eLoadClose OF
			E_LoadClose.None:
				CASE _eLoadClass OF
					E_LoadClass.Acquire:
						IF GVL.stHandshake.bLine1ToAcquire AND _station.iStepNow=_station.iStepNext  THEN
							_station.iStepNext:=1301;
						END_IF
						IF GVL.stHandshake.bBufferToAcquire AND _station.iStepNow=_station.iStepNext THEN
							_station.iStepNext:=1251;
						END_IF
					E_LoadClass.Line0,E_LoadClass.None:
						IF GVL.stHandshake.bBufferToAcquire AND _station.iStepNow=_station.iStepNext THEN
							_station.iStepNext:=1251;
						END_IF
						IF GVL.stHandshake.bLine1ToAcquire AND _station.iStepNow=_station.iStepNext THEN
							_station.iStepNext:=1301;
						END_IF
					E_LoadClass.Sensor:						
						IF GVL.stSetting.bLine0Priority THEN
							IF GVL.stHandshake.bBufferToAcquire AND _station.iStepNow=_station.iStepNext THEN
								_station.iStepNext:=1251;
							END_IF
							//IF GVL.stHandshake.bLine1ToAcquire AND _station.iStepNow=_station.iStepNext THEN
							//	_station.iStepNext:=1301;
							//END_IF
						ELSE
							IF GVL.stHandshake.bLine1ToAcquire AND _station.iStepNow=_station.iStepNext  THEN
								_station.iStepNext:=1301;
							END_IF
							IF GVL.stHandshake.bBufferToAcquire AND _station.iStepNow=_station.iStepNext THEN
								_station.iStepNext:=1251;
							END_IF
						END_IF			
				END_CASE
			E_LoadClose.Acquire:
				IF GVL.stHandshake.bBufferToAcquire THEN
					_station.iStepNext:=1251;
				END_IF
			E_LoadClose.Line0:
				IF GVL.I.bAcquireCheck0 OR GVL.I.bAcquireCheck1 THEN
					_station.iStepNext:=1301;
				END_IF
		END_CASE
	1251:
		_station.arrInfo[E_Language.Chinese]:="等待拨料升降气缸至缩回位";
		IF G_arrCylinder[E_Cylinder.AcquireElevator].stStatus.bHomeDone THEN
			GVL.stHandshake.bAcquireToBuffer:=TRUE;
			_station.iStepNext:=1261;
		END_IF
	1261:
		_station.arrInfo[E_Language.Chinese]:="等待复位请求信号";
		IF NOT GVL.stHandshake.bBufferToAcquire THEN
			GVL.stHandshake.bAcquireToBuffer:=FALSE;
			_station.iStepNext:=1801;
		END_IF
	1301:
		_station.arrInfo[E_Language.Chinese]:="顶升气缸缩回";		
		IF  G_arrFbCylinder[E_Cylinder.AcquireLift].M_HomeRequest() THEN
			GVL.stHandshake.bAcquireToLine1:=TRUE;
			_station.iStepNext:=1311;
		END_IF	
	1311:	
		_station.arrInfo[E_Language.Chinese]:="等待产品到位";
		GVL.stOverTime.bAcquireCheck2:=TRUE;
		IF GVL.I.bAcquireCheck2 THEN
			GVL.stOverTime.bAcquireCheck2:=FALSE;
			_station.iStepNext:=1321;
		END_IF
	1321:
		_station.arrInfo[E_Language.Chinese]:="等待接驳线复位接驳站收料请求";
		GVL.stHandshake.bAcquireToLine1:=FALSE;
		IF NOT GVL.stHandshake.bLine1ToAcquire THEN
			_station.iStepNext:=1701;
		END_IF
	1701:
		_station.arrInfo[E_Language.Chinese]:="判断拨料气缸 升降气缸 是否到位";
		IF G_arrCylinder[E_Cylinder.AcquireElevator].stStatus.bHomeDone AND G_arrCylinder[E_Cylinder.AcquirePush].stStatus.bWorkDone THEN
			_station.iStepNext:=1751;
		END_IF
	1751:
		_station.arrInfo[E_Language.Chinese]:="顶升气缸伸出 升降气缸伸出";
		IF  G_arrFbCylinder[E_Cylinder.AcquireLift].M_WorkRequest() AND G_arrFbCylinder[E_Cylinder.AcquireElevator].M_WorkRequest() THEN 
			_station.iStepNext:=1801;
		END_IF	
	1801:
		_station.arrInfo[E_Language.Chinese]:="升降气缸伸出";
		// 等待拨料气缸 至后位 再伸出
		IF G_arrCylinder[E_Cylinder.AcquirePush].stStatus.bWorkDone THEN
			IF G_arrFbCylinder[E_Cylinder.AcquireElevator].M_WorkRequest() THEN
				_station.iStepNext:=1901;
			END_IF
		END_IF		
	1901:
		_station.arrInfo[E_Language.Chinese]:="等待转向站请求放料";
		IF GVL.stHandshake.bSteering THEN
			GVL.stHandshake.bSteeringOk:=TRUE;
			_station.iStepNext:=2001;
		END_IF
	2001:
		_station.arrInfo[E_Language.Chinese]:="拨料气缸至前位";
		IF G_arrFbCylinder[E_Cylinder.AcquirePush].M_HomeRequest() THEN
			_station.iStepNext:=2101;
		END_IF
	2101:
		_station.arrInfo[E_Language.Chinese]:="等待复位请求信号";
		IF NOT GVL.stHandshake.bSteering THEN
			GVL.stHandshake.bSteeringOk:=FALSE;
			_station.iStepNext:=2201;
		END_IF
	2201:
		_station.arrInfo[E_Language.Chinese]:="拨料气缸至后位 升降气缸缩回";
		G_arrFbCylinder[E_Cylinder.AcquirePush].M_WorkRequest();
		G_arrFbCylinder[E_Cylinder.AcquireElevator].M_HomeRequest();
		_station.iStepNext:=1100;
END_CASE
END_ACTION

ACTION A_Home:
CASE _station.iStepNow OF
	0:
		_station.arrInfo[E_Language.Chinese]:="等待初始化";
		_station.iStepNext:=SEL(_bEnable,1000,100);
	100:
		_station.arrInfo[E_Language.Chinese]:="前阻挡气缸伸出";
		IF G_arrFbCylinder[E_Cylinder.AcquirePrevent0].M_WorkRequest() THEN
			IF GVL.stSetting.bAcquirePrevent2Shield THEN
				_station.iStepNext:=200;
			ELSE
				_station.iStepNext:=110;
			END_IF	
		END_IF
	110:
		_station.arrInfo[E_Language.Chinese]:="前前阻挡气缸缩回";
		IF G_arrFbCylinder[E_Cylinder.AcquirePrevent2].M_HomeRequest() THEN
			_station.iStepNext:=200;
		END_IF			
	200:
		_station.arrInfo[E_Language.Chinese]:="后阻挡气缸伸出";
		IF G_arrFbCylinder[E_Cylinder.AcquirePrevent1].M_WorkRequest() THEN
			_station.iStepNext:=300;
		END_IF
	300:
		_station.arrInfo[E_Language.Chinese]:="升降气缸缩回";
		IF  G_arrFbCylinder[E_Cylinder.AcquireElevator].M_HomeRequest() THEN
			_station.iStepNext:=400;
		END_IF
	400:
		_station.arrInfo[E_Language.Chinese]:="拨料气缸至后位";
		IF  G_arrFbCylinder[E_Cylinder.AcquirePush].M_WorkRequest() THEN
			_station.iStepNext:=500;
		END_IF
	500:
		_station.arrInfo[E_Language.Chinese]:="顶升气缸伸出";
		IF G_arrFbCylinder[E_Cylinder.AcquireLift].M_WorkRequest() THEN
			_station.iStepNext:=1000;
		END_IF
END_CASE
END_ACTION

END_PROGRAM

// ---- POUs/P_StationLine0Buffer.TcPOU
PROGRAM P_StationLine0Buffer
VAR
	_station:					REFERENCE TO ST_SystemStation;
	_bEnable: 					BOOL;
END_VAR

_station REF= G_arrStation[E_Station.Line0Buffer];
_station.arrName[E_Language.Chinese]:="线体0上料缓存";
_station.arrName[E_Language.Vietnamese]:="Bộ nhớ nhớ dòng chính";
_bEnable:= NOT GVL.stSetting.arrStationShield[E_Station.Line0Buffer];
GVL.stSetting.arrStationShield[E_Station.Line0Buffer]:=GVL.stSetting.bManualLoad;


A_Home();
A_Auto();

ACTION A_Auto:
CASE _station.iStepNow OF
	1000:
		_station.arrInfo[E_Language.Chinese]:="初始化完成等待启动";
		IF _bEnable  THEN
			_station.iStepNext:=1101;
		END_IF
	1101:
		_station.arrInfo[E_Language.Chinese]:="判断缓存站是否有料";
		
		IF NOT GVL.stSetting.bLine0BufferShield THEN
			IF GVL.I.bLine0Check3 THEN
				_station.iStepNext:=1501;
			ELSE
				_station.iStepNext:=1201;
			END_IF
		ELSE
			IF GVL.I.bLine0Check3 THEN
				_station.iStepNext:=1501;
			END_IF
		END_IF
		
	1201:
		_station.arrInfo[E_Language.Chinese]:="请求上料站放料";
		GVL.stHandshake.bBufferToLoad:=TRUE;
		IF GVL.stHandshake.bLoadToBuffer THEN
			_station.iStepNext:=1301;
		END_IF
	1301:
		_station.arrInfo[E_Language.Chinese]:="等待产品到位";
		GVL.stOverTime.bLine0Check3:=TRUE;
		IF GVL.I.bLine0Check3 THEN
			GVL.stOverTime.bLine0Check3:=FALSE;
			_station.iStepNext:=1401;
		END_IF
	1401:
		_station.arrInfo[E_Language.Chinese]:="复位请求放料信号";
		GVL.stHandshake.bBufferToLoad:=FALSE;
		IF NOT GVL.stHandshake.bLoadToBuffer THEN
			_station.iStepNext:=1501;
		END_IF	
	1501:
		_station.arrInfo[E_Language.Chinese]:="请求放料";
		CASE GVL_Data.stRecipe.eMachineType OF
			 E_MachineType._367:
				IF GVL.stHandshake.bSteering THEN
					GVL.stHandshake.bSteeringOk:=TRUE;
					_station.iStepNext:=1801;
				END_IF
			ELSE
				GVL.stHandshake.bBufferToAcquire:=TRUE;
		 		IF GVL.stHandshake.bAcquireToBuffer THEN
				 _station.iStepNext:=1812;
		 		END_IF
		END_CASE
	1801:
		_station.arrInfo[E_Language.Chinese]:="拨料气缸至工作位";
		G_arrFbCylinder[E_Cylinder.Line0Push].M_HomeRequest();
		IF NOT GVL.I.bLine0Push_Cyl_W THEN
			_station.iStepNext:=1802;
		END_IF	
	1802:
		_station.arrInfo[E_Language.Chinese]:="请求主流线上料";
		IF GVL.I.bLine0Push_Cyl_Safe OR GVL.I.bLine0Push_Cyl_H THEN
			GVL.stHandshake.bBufferToLoad:=TRUE;
			_station.iStepNext:=1811;
		END_IF		
	1811:
		_station.arrInfo[E_Language.Chinese]:="拨料气缸至工作位";
		IF G_arrFbCylinder[E_Cylinder.Line0Push].M_HomeRequest() THEN
			_station.iStepNext:=1821;
		END_IF
	1812:
		_station.arrInfo[E_Language.Chinese]:="拨料气缸至工作位";
		IF G_arrFbCylinder[E_Cylinder.Line0Push].M_HomeRequest() THEN
			_station.iStepNext:=1821;
		END_IF	
	1821:
	    G_arrFbCylinder[E_Cylinder.Line0Push].M_WorkRequest();
		IF NOT GVL.I.bLine0Push_Cyl_H THEN  
			_station.iStepNext:=1831;
		END_IF 
	1831:
		_station.arrInfo[E_Language.Chinese]:="等待放料结束";
		
		CASE GVL_Data.stRecipe.eMachineType OF
			E_MachineType._367:
			
				G_arrFbCylinder[E_Cylinder.Line0PushElevator].M_HomeRequest();
				
				IF (GVL.I.bLine0Push_Cyl_Safe OR GVL.I.bLine0Push_Cyl_W) AND NOT GVL.I.bLine0PushElevator_Cyl_H THEN
					_station.iStepNext:=2001;	
				END_IF
				
				IF NOT GVL.stHandshake.bSteering THEN
					GVL.stHandshake.bSteeringOk:=FALSE;
					_station.iStepNext:=1851;
				END_IF
				
				
			ELSE
				GVL.stHandshake.bBufferToAcquire:=FALSE;
				IF NOT GVL.stHandshake.bAcquireToBuffer THEN
					_station.iStepNext:=1901;
				END_IF
		END_CASE
	1851:
		_station.arrInfo[E_Language.Chinese]:="拨料气缸至待料位 拨料升降气缸至上升位";
		
		IF (GVL.I.bLine0Push_Cyl_Safe OR GVL.I.bLine0Push_Cyl_W) AND NOT GVL.I.bLine0PushElevator_Cyl_H THEN
			_station.iStepNext:=2001;	
		END_IF	
		
		IF G_arrFbCylinder[E_Cylinder.Line0Push].M_WorkRequest() AND G_arrFbCylinder[E_Cylinder.Line0PushElevator].M_HomeRequest() THEN
			_station.iStepNext:=1861;
		END_IF
	1861:
		_station.arrInfo[E_Language.Chinese]:="拨料升降气缸至下降位";
		IF G_arrFbCylinder[E_Cylinder.Line0PushElevator].M_WorkRequest() THEN
			_station.iStepNext:=1201;
		END_IF		
	1901:
		_station.arrInfo[E_Language.Chinese]:="拨料气缸至待料位";
		IF G_arrFbCylinder[E_Cylinder.Line0Push].M_WorkRequest() THEN
			_station.iStepNext:=1101;
		END_IF				
	2001:
		_station.arrInfo[E_Language.Chinese]:="拨料气缸至工作位 拨料升降气缸至上升位";
		IF G_arrFbCylinder[E_Cylinder.Line0Push].M_HomeRequest() AND G_arrFbCylinder[E_Cylinder.Line0PushElevator].M_HomeRequest() THEN
			_station.iStepNext:=2101;
		END_IF
	2101:		
		_station.arrInfo[E_Language.Chinese]:="拨料升降气缸上升速度过慢报警";
		IF NOT GVL.AlarmResetMark THEN
			GVL.stOverTime.bLine0PushElevatorUp:=TRUE;
		ELSE
			_station.iStepNext:=2201;
		END_IF		
	2201:
		GVL.stOverTime.bLine0PushElevatorUp:=FALSE;
		GVL.AlarmResetMark:=FALSE;
		IF NOT GVL.stOverTime.bLine0PushElevatorUp THEN
			_station.iStepNext:=1821;
		END_IF		
		
END_CASE
END_ACTION

ACTION A_Home:
CASE _station.iStepNow OF
	0:
		_station.arrInfo[E_Language.Chinese]:="等待初始化";
		_station.iStepNext:=SEL(_bEnable,1000,100);	
	100:
		_station.arrInfo[E_Language.Chinese]:="判断拆解机机型";
		_station.iStepNext:=SEL(GVL_Data.stRecipe.eMachineType=E_MachineType._367,400,200);			
	200:
		_station.arrInfo[E_Language.Chinese]:="判断拨料气缸位置";
		IF GVL.I.bLine0Push_Cyl_H THEN
			_station.iStepNext:=210;
		ELSIF GVL.I.bLine0Push_Cyl_W THEN 
			_station.iStepNext:=400;
		ELSE
			_station.iStepNext:=300;
		END_IF	
	210:		
		_station.arrInfo[E_Language.Chinese]:="拨料气缸至待料位";
	    G_arrFbCylinder[E_Cylinder.Line0Push].M_WorkRequest();
		IF NOT GVL.I.bLine0Push_Cyl_H THEN
			_station.iStepNext:=220;
		END_IF				
	220:
		_station.arrInfo[E_Language.Chinese]:="拨料升降气缸至上升位";
		IF G_arrFbCylinder[E_Cylinder.Line0Push].M_WorkRequest() AND G_arrFbCylinder[E_Cylinder.Line0PushElevator].M_HomeRequest() THEN
			_station.iStepNext:=500;
		END_IF	
	300:
		_station.arrInfo[E_Language.Chinese]:="拨料升降气缸至上升位";
		IF G_arrFbCylinder[E_Cylinder.Line0PushElevator].M_HomeRequest() THEN
			_station.iStepNext:=400;
		END_IF		
	400:
		_station.arrInfo[E_Language.Chinese]:="拨料气缸至待料位";
		IF G_arrFbCylinder[E_Cylinder.Line0Push].M_WorkRequest() THEN
			_station.iStepNext:=SEL(GVL_Data.stRecipe.eMachineType=E_MachineType._367,1000,500);
		END_IF
	500:
		_station.arrInfo[E_Language.Chinese]:="拨料升降气缸至下降位";
		IF G_arrFbCylinder[E_Cylinder.Line0PushElevator].M_WorkRequest() THEN
			_station.iStepNext:=1000;
		END_IF	
		
		
		
END_CASE
END_ACTION

END_PROGRAM

// ---- POUs/P_StationLine0Load.TcPOU
PROGRAM P_StationLine0Load
VAR
	_station:					REFERence TO ST_SystemStation;
	_bEnable: 					BOOL;
	_stHandshake:				ST_Handshake;
	_stTimeOut:                 ST_TimeOut;
END_VAR

_station REF= G_arrStation[E_Station.Line0Load];
_station.arrName[E_Language.Chinese]:="线条0上料站";
_station.arrName[E_Language.Vietnamese]:="Dòng trực tuyến";
_bEnable:= NOT GVL.stSetting.arrStationShield[E_Station.Line0Load];
GVL.stSetting.arrStationShield[E_Station.Line0Load]:=GVL.stSetting.bManualLoad;


A_Home();
A_Auto();

ACTION A_Auto:
CASE _station.iStepNow OF
	1000:
		_station.arrInfo[E_Language.Chinese]:="初始化完成等待启动";
		IF _bEnable  THEN
			_station.iStepNext:=1100;
		END_IF
	1100:
		_station.arrInfo[E_Language.Chinese]:="判断阻挡位是否有料";
		IF GVL.I.bLine0Check2 THEN
			_station.iStepNext:=1451;
		END_IF		
	1451:
		_station.arrInfo[E_Language.Chinese]:="分料气缸伸出";
		IF G_arrFbCylinder[E_Cylinder.Line0Part].M_WorkRequest() THEN
			_station.iStepNext:=1501;
		END_IF
	1501:
		_station.arrInfo[E_Language.Chinese]:="等待缓存站请求放料";
		IF GVL.stHandshake.bBufferToLoad THEN
			GVL.stHandshake.bLoadToBuffer:=TRUE;
			_station.iStepNext:=1601;
		END_IF
	1601:
		_station.arrInfo[E_Language.Chinese]:="阻挡气缸缩回";
		IF G_arrFbCylinder[E_Cylinder.Line0Prevent].M_HomeRequest() THEN
			_station.iStepNext:=1701;
		END_IF	
	1701:
		_station.arrInfo[E_Language.Chinese]:="等待托盘流出";
		IF NOT GVL.I.bLine0Check2 THEN
			_station.iStepNext:=1711;
		END_IF
	1711:
		_station.arrInfo[E_Language.Chinese]:="等待产品到位";
		GVL.stOverTime.bLine0Check3:=TRUE;
		IF GVL.I.bLine0Check3 THEN
			GVL.stOverTime.bLine0Check3:=FALSE;
			_station.iStepNext:=1901;
		END_IF
	1901:
		_station.arrInfo[E_Language.Chinese]:="阻挡气缸伸出";
		IF G_arrFbCylinder[E_Cylinder.Line0Prevent].M_WorkRequest() THEN	
			_station.iStepNext:=1911;
		END_IF
	1911:		
		_station.arrInfo[E_Language.Chinese]:="分料气缸缩回";
		IF G_arrFbCylinder[E_Cylinder.Line0Part].M_HomeRequest() THEN
			_station.iStepNext:=1921;
		END_IF
	1921:
		_station.arrInfo[E_Language.Chinese]:="等待复位请求信号";
		IF NOT GVL.stHandshake.bBufferToLoad THEN
			GVL.stHandshake.bLoadToBuffer:=FALSE;
			_station.iStepNext:=1100;
		END_IF			
	
END_CASE
END_ACTION

ACTION A_Home:
CASE _station.iStepNow OF
	0:
		_station.arrInfo[E_Language.Chinese]:="等待初始化";
		GVL.stHandshake:=_stHandshake;
		GVL.stOverTime:=_stTimeOut;
		_station.iStepNext:=SEL(_bEnable,1000,100);
	100:
		_station.arrInfo[E_Language.Chinese]:="阻挡气缸伸出";
		IF  G_arrFbCylinder[E_Cylinder.Line0Prevent].M_WorkRequest() THEN
			_station.iStepNext:=200;
		END_IF
	200:
		_station.arrInfo[E_Language.Chinese]:="分料气缸缩回";
		IF  G_arrFbCylinder[E_Cylinder.Line0Part].M_HomeRequest() THEN
			_station.iStepNext:=1000;
		END_IF
END_CASE
END_ACTION

END_PROGRAM

// ---- POUs/P_StationOpenLock.TcPOU
PROGRAM P_StationOpenLock
VAR
	_station:					REFERence TO ST_SystemStation;
	_bEnable: 					BOOL;
	_OpenLockCheck0FTrig:       Tc2_Standard.F_TRIG;
END_VAR

_station REF= G_arrStation[E_Station.OpenLock];
_station.arrName[E_Language.Chinese]:="解锁站";
_station.arrName[E_Language.Vietnamese]:="Mở khóa nhà ga";
_bEnable:=NOT GVL.stSetting.arrStationShield[E_Station.OpenLock];

IF GVL_Data.stRecipe.eMachineType=E_MachineType._311 THEN
	A_Home311();
	A_Auto311();
ELSE
	A_Home();
	A_Auto();
END_IF

_OpenLockCheck0FTrig(CLK:= GVL.I.bOpenLockCheck0, Q=> );

GVL._arrAutoTimer[E_Timer.SteeringCheck1F](IN:=NOT GVL.I.bSteeringCheck1 AND GVL.I.bSteeringAcquireElevator_Cyl_H, PT:=TO_TIME(GVL_Data.stRecipe.arrAutoTon[E_Timer.SteeringCheck1F]), Q=>GVL._arrAutoTimerOut[E_Timer.SteeringCheck1F] , ET=> );

ACTION A_Auto:
CASE _station.iStepNow OF
	1000:
		_station.arrInfo[E_Language.Chinese]:="初始化完成等待启动";
		IF _bEnable THEN
			_station.iStepNext:=1101;
		END_IF
	1101:
		_station.arrInfo[E_Language.Chinese]:="判断是否有料";
		IF NOT GVL.I.bOpenLockCheck THEN
			_station.iStepNext:=1201;
		END_IF
	1201:
		_station.arrInfo[E_Language.Chinese]:="请求上料";
		GVL.stHandshake.bOpenToSteering:=TRUE;
		IF GVL.stHandshake.bSteeringToOpen THEN
			_station.iStepNext:=1301;
		END_IF
	1301:
		_station.arrInfo[E_Language.Chinese]:="等待产品从旋转站流出";
		GVL.stOverTime.bOpenLockCheck:=TRUE;
		IF GVL._arrAutoTimerOut[E_Timer.SteeringCheck1F] THEN
			GVL.stOverTime.bOpenLockCheck:=FALSE;
			_station.iStepNext:=1401;//解锁站流入传感器安装后改为 1311
		END_IF
	1311:		
		_station.arrInfo[E_Language.Chinese]:="产品从旋转站流出确认";
		IF _OpenLockCheck0FTrig.Q THEN
			_station.iStepNext:=1401;
		END_IF	
	1401:
		_station.arrInfo[E_Language.Chinese]:="复位上料请求";
		GVL.stHandshake.bOpenToSteering:=FALSE;
		IF  NOT GVL.stHandshake.bSteeringToOpen THEN
			_station.iStepNext:=1411;
		END_IF
	1411:
		_station.arrInfo[E_Language.Chinese]:="等待产品到位";
		GVL.stOverTime.bOpenLockCheck:=TRUE;
		IF GVL.I.bOpenLockCheck THEN
			GVL.stOverTime.bOpenLockCheck:=FALSE;
			_station.iStepNext:=1501;
		END_IF			
	1501:
		_station.arrInfo[E_Language.Chinese]:="顶升气缸伸出";
		IF G_arrFbCylinder[E_Cylinder.OpenLockLift].M_WorkRequest() THEN
			IF GVL_Data.stRecipe.eMachineType=E_MachineType._373 AND NOT GVL.stSetting.bOpenLockPressShield THEN 
				_station.iStepNext:=1511;
			ELSE
			_station.iStepNext:=1601;
			END_IF
		END_IF
	1511:	
		_station.arrInfo[E_Language.Chinese]:="解压侧推气缸伸出";	
		IF G_arrFbCylinder[E_Cylinder.OpenLockPressPush].M_WorkRequest() THEN
			_station.iStepNext:=1521;
		END_IF
	1521:	
		_station.arrInfo[E_Language.Chinese]:="解压旋转气缸旋转";	
		IF G_arrFbCylinder[E_Cylinder.OpenLockPressRotate].M_WorkRequest() THEN
			_station.iStepNext:=1531;
		END_IF	
	1531:	
		_station.arrInfo[E_Language.Chinese]:="解压旋转气缸返回";	
		IF G_arrFbCylinder[E_Cylinder.OpenLockPressRotate].M_HomeRequest() THEN
			_station.iStepNext:=1541;		
		END_IF		
	1541:
		_station.arrInfo[E_Language.Chinese]:="解压侧推气缸缩回 侧推气缸伸出";
		IF M_PushWork() AND G_arrFbCylinder[E_Cylinder.OpenLockPressPush].M_HomeRequest() THEN
			_station.iStepNext:=1701;
		END_IF		
	1601:
		_station.arrInfo[E_Language.Chinese]:="侧推气缸伸出";
		IF M_PushWork() THEN
			_station.iStepNext:=1701;
		END_IF
	1701:
		_station.arrInfo[E_Language.Chinese]:="旋转气缸至右位 校平气缸伸出";
		IF G_arrFbCylinder[E_Cylinder.OpenLockRotate].M_WorkRequest() AND M_StandardWork() THEN
			_station.iStepNext:=1801;
		END_IF
	1801:
		_station.arrInfo[E_Language.Chinese]:="侧推气缸缩回 校平气缸缩回 阻挡气缸缩回";
		IF M_PushHome() AND M_StandardHome()  AND  G_arrFbCylinder[E_Cylinder.OpenLockPrevent].M_HomeRequest() THEN
           _station.iStepNext:=2001;
		END_IF
	2001:
		_station.arrInfo[E_Language.Chinese]:="等待取Uc站请求放料";
		IF GVL.stHandshake.bTakeUcToOpen THEN
			GVL.stHandshake.bOpenToTakeUc:=TRUE;
			GVL.stHandshake.bOpenToSteering:=TRUE;//同时请求旋转站放料
			_station.iStepNext:=2101;
		END_IF
	2101:
	     _station.arrInfo[E_Language.Chinese]:="顶升气缸下降,解锁旋转气缸至左位";
		IF G_arrFbCylinder[E_Cylinder.OpenLockLift].M_HomeRequest() AND G_arrFbCylinder[E_Cylinder.OpenLockRotate].M_HomeRequest() THEN
			_station.iStepNext:=2201;
		END_IF
	2201:
		_station.arrInfo[E_Language.Chinese]:="等待复位请求信号";
		IF NOT GVL.stHandshake.bTakeUcToOpen THEN
			GVL.stHandshake.bOpenToTakeUc:=FALSE;
			_station.iStepNext:=2301;
		END_IF		
	2301:
		_station.arrInfo[E_Language.Chinese]:="阻挡气缸伸出";
		IF G_arrFbCylinder[E_Cylinder.OpenLockPrevent].M_WorkRequest() THEN
			_station.iStepNext:=1201;
		END_IF		

END_CASE
END_ACTION

ACTION A_Auto311:
CASE _station.iStepNow OF
	1000:
		_station.arrInfo[E_Language.Chinese]:="初始化完成等待启动";
		IF _bEnable THEN
			_station.iStepNext:=1101;
		END_IF
	1101:
		_station.arrInfo[E_Language.Chinese]:="判断是否有料";
		IF NOT GVL.I.bOpenLockCheck THEN
			_station.iStepNext:=1201;
		END_IF
	1201:
		_station.arrInfo[E_Language.Chinese]:="请求上料";
		GVL.stHandshake.bOpenToSteering:=TRUE;
		IF GVL.stHandshake.bSteeringToOpen THEN
			_station.iStepNext:=1301;
		END_IF
	1301:
		_station.arrInfo[E_Language.Chinese]:="等待产品从旋转站流出";
		GVL.stOverTime.bOpenLockCheck:=TRUE;
		IF GVL._arrAutoTimerOut[E_Timer.SteeringCheck1F] THEN
			GVL.stOverTime.bOpenLockCheck:=FALSE;
			_station.iStepNext:=1401;//传感器安装后改为 1311
		END_IF
	1311:		
		_station.arrInfo[E_Language.Chinese]:="产品从旋转站流出确认";
		IF _OpenLockCheck0FTrig.Q THEN
			_station.iStepNext:=1401;
		END_IF			
	1401:
		_station.arrInfo[E_Language.Chinese]:="复位上料请求";
		GVL.stHandshake.bOpenToSteering:=FALSE;
		IF  NOT GVL.stHandshake.bSteeringToOpen THEN
			_station.iStepNext:=1411;
		END_IF
	1411:
		_station.arrInfo[E_Language.Chinese]:="等待产品到位";
		GVL.stOverTime.bOpenLockCheck:=TRUE;
		IF GVL.I.bOpenLockCheck THEN
			GVL.stOverTime.bOpenLockCheck:=FALSE;
			_station.iStepNext:=1501;
		END_IF			
	1501:
		_station.arrInfo[E_Language.Chinese]:="顶升气缸伸出";
		IF G_arrFbCylinder[E_Cylinder.OpenLockLift].M_WorkRequest() THEN
			_station.iStepNext:=1511;
		END_IF
	1511:		
		_station.arrInfo[E_Language.Chinese]:="检测工装有无误合盖";
		IF GVL.I.bFrockCloseCheck OR GVL.stSetting.bFrockCloseCheckShield THEN
			_station.iStepNext:=1601;
		ELSE
			_station.iStepNext:=1521;
		END_IF
	1521:	
		_station.arrInfo[E_Language.Chinese]:="置位工装检测失败记忆";
		GVL.TakeUcSafeCheckNG_OpenLock:=TRUE;
		IF GVL.TakeUcSafeCheckNG_OpenLock THEN
			_station.iStepNext:=2001;
		END_IF		
	1601:
		_station.arrInfo[E_Language.Chinese]:="升降气缸缩回";
		GVL.TakeUcSafeCheckNG_OpenLock:=FALSE;
		IF G_arrFbCylinder[E_Cylinder.OpenLockElevator].M_HomeRequest() THEN
			_station.iStepNext:=1701;
		END_IF
	1701:
		_station.arrInfo[E_Language.Chinese]:="按压气缸伸出";
		IF G_arrFbCylinder[E_Cylinder.OpenLockPin].M_WorkRequest() THEN
			_station.iStepNext:=1801;
		END_IF
	1801:
		_station.arrInfo[E_Language.Chinese]:="平移气缸缩回";
		IF G_arrFbCylinder[E_Cylinder.OpenLockTranslation].M_HomeRequest() THEN
			_station.iStepNext:=1901;
		END_IF
	1901:
		_station.arrInfo[E_Language.Chinese]:="旋转气缸至初始位";
		IF G_arrFbCylinder[E_Cylinder.OpenLockRotate].M_HomeRequest() THEN
			_station.iStepNext:=1951;
		END_IF
	1951:
		_station.arrInfo[E_Language.Chinese]:="升降气缸伸出 按压气缸缩回";
		IF G_arrFbCylinder[E_Cylinder.OpenLockElevator].M_WorkRequest() AND G_arrFbCylinder[E_Cylinder.OpenLockPin].M_HomeRequest()  THEN
			_station.iStepNext:=2001;
		END_IF
	2001:
		_station.arrInfo[E_Language.Chinese]:="等待取Uc站请求放料";
		IF GVL.stHandshake.bTakeUcToOpen THEN
			GVL.stHandshake.bOpenToTakeUc:=TRUE;
			GVL.stHandshake.bOpenToSteering:=TRUE;//同时请求旋转站放料
			_station.iStepNext:=2051;
		END_IF
	2051:
		_station.arrInfo[E_Language.Chinese]:="顶升气缸缩回 阻挡气缸缩回";
		IF G_arrFbCylinder[E_Cylinder.OpenLockPrevent].M_HomeRequest() AND G_arrFbCylinder[E_Cylinder.OpenLockLift].M_HomeRequest() THEN
			_station.iStepNext:=2101;
		END_IF
	2101:
		_station.arrInfo[E_Language.Chinese]:="旋转气缸至工作位 平移气缸伸出";
		G_arrFbCylinder[E_Cylinder.OpenLockRotate].M_WorkRequest();
		G_arrFbCylinder[E_Cylinder.OpenLockTranslation].M_WorkRequest();
		_station.iStepNext:=2201;		
	2201:
		_station.arrInfo[E_Language.Chinese]:="等待复位请求信号";
		IF NOT GVL.stHandshake.bTakeUcToOpen THEN
			GVL.stHandshake.bOpenToTakeUc:=FALSE;
			_station.iStepNext:=2301;
		END_IF
	2301:
		_station.arrInfo[E_Language.Chinese]:="阻挡气缸伸出";
		IF G_arrFbCylinder[E_Cylinder.OpenLockPrevent].M_WorkRequest() AND G_arrFbCylinder[E_Cylinder.OpenLockRotate].M_WorkRequest() AND G_arrFbCylinder[E_Cylinder.OpenLockTranslation].M_WorkRequest() THEN
			_station.iStepNext:=1201;
		END_IF

END_CASE
END_ACTION

ACTION A_Home:
CASE _station.iStepNow OF
	0:
		_station.arrInfo[E_Language.Chinese]:="等待初始化";
		_station.iStepNext:=SEL(_bEnable,1000,100);
	100:		
		IF GVL_Data.stRecipe.eMachineType=E_MachineType._373 AND NOT GVL.stSetting.bOpenLockPressShield THEN 
			_station.iStepNext:=110;
		ELSE
			_station.iStepNext:=150;
		END_IF		
	110:
		_station.arrInfo[E_Language.Chinese]:="解压旋转气缸返回";
		IF G_arrFbCylinder[E_Cylinder.OpenLockPressRotate].M_HomeRequest() THEN
			_station.iStepNext:=120;
		END_IF	
	120:
		_station.arrInfo[E_Language.Chinese]:="解压侧推气缸缩回";
		IF G_arrFbCylinder[E_Cylinder.OpenLockPressPush].M_HomeRequest() THEN
			_station.iStepNext:=150;
		END_IF	
	150:	
		_station.arrInfo[E_Language.Chinese]:="侧推气缸缩回";
		IF M_PushHome() THEN
			_station.iStepNext:=200;
		END_IF
	200:
		_station.arrInfo[E_Language.Chinese]:="旋转气缸至左位";
		IF G_arrFbCylinder[E_Cylinder.OpenLockRotate].M_HomeRequest() THEN
			_station.iStepNext:=300;
		END_IF
	300:
		_station.arrInfo[E_Language.Chinese]:="阻挡气缸伸出";
		IF G_arrFbCylinder[E_Cylinder.OpenLockPrevent].M_WorkRequest() THEN
			_station.iStepNext:=400;
		END_IF
	400:
		_station.arrInfo[E_Language.Chinese]:="顶升气缸缩回";
		IF G_arrFbCylinder[E_Cylinder.OpenLockLift].M_HomeRequest() THEN
			_station.iStepNext:=500;
		END_IF
	500:
		_station.arrInfo[E_Language.Chinese]:="校平气缸缩回";
		IF  M_StandardHome() THEN
			_station.iStepNext:=1000;
		END_IF
END_CASE
END_ACTION

ACTION A_Home311:
CASE _station.iStepNow OF
	0:
		_station.arrInfo[E_Language.Chinese]:="等待初始化";
		_station.iStepNext:=SEL(_bEnable,1000,100);
	100:
		_station.arrInfo[E_Language.Chinese]:="升降气缸伸出";
		IF 	G_arrFbCylinder[E_Cylinder.OpenLockElevator].M_WorkRequest() THEN
			_station.iStepNext:=150;
		END_IF
	150:
		_station.arrInfo[E_Language.Chinese]:="按压气缸缩回";
		IF G_arrFbCylinder[E_Cylinder.OpenLockPin].M_HomeRequest() THEN
			_station.iStepNext:=200;
		END_IF
	200:
		_station.arrInfo[E_Language.Chinese]:="旋转气缸至工作位";
		IF G_arrFbCylinder[E_Cylinder.OpenLockRotate].M_WorkRequest() THEN
			_station.iStepNext:=300;
		END_IF
	300:
		_station.arrInfo[E_Language.Chinese]:="平移气缸伸出";
		IF 	G_arrFbCylinder[E_Cylinder.OpenLockTranslation].M_WorkRequest() THEN
			_station.iStepNext:=500;
		END_IF
	500:
		_station.arrInfo[E_Language.Chinese]:="阻挡气缸伸出";
		IF G_arrFbCylinder[E_Cylinder.OpenLockPrevent].M_WorkRequest() THEN
			_station.iStepNext:=600;
		END_IF
	600:
		_station.arrInfo[E_Language.Chinese]:="顶升气缸缩回";
		IF G_arrFbCylinder[E_Cylinder.OpenLockLift].M_HomeRequest() THEN
			_station.iStepNext:=1000;
		END_IF
END_CASE
END_ACTION

METHOD M_PushHome : BOOL
VAR_INPUT
END_VAR
CASE GVL_Data.stRecipe.eMachineType OF
	E_MachineType._200,E_MachineType._069,E_MachineType._367:
		M_PushHome:=G_arrFbCylinder[E_Cylinder.OpenLockPush].M_HomeRequest() AND G_arrFbCylinder[E_Cylinder.OpenLockPush2].M_HomeRequest();
	E_MachineType._373:
		M_PushHome:=G_arrFbCylinder[E_Cylinder.OpenLockPush].M_HomeRequest();
END_CASE
END_METHOD

METHOD M_PushWork : BOOL
VAR_INPUT
END_VAR
CASE GVL_Data.stRecipe.eMachineType OF
	E_MachineType._200,E_MachineType._069,E_MachineType._367:
		M_PushWork:=G_arrFbCylinder[E_Cylinder.OpenLockPush].M_WorkRequest() AND G_arrFbCylinder[E_Cylinder.OpenLockPush2].M_WorkRequest();
	E_MachineType._373:
		M_PushWork:=G_arrFbCylinder[E_Cylinder.OpenLockPush].M_WorkRequest();
END_CASE
END_METHOD

METHOD M_StandardHome : BOOL
VAR_INPUT
END_VAR
M_StandardHome:=TRUE;
END_METHOD

METHOD M_StandardWork : BOOL
VAR_INPUT
END_VAR
M_StandardWork:=TRUE;
END_METHOD

END_PROGRAM

// ---- POUs/P_StationTakeUc.TcPOU
PROGRAM P_StationTakeUc
VAR
	_station:					REFERENCE TO ST_SystemStation;
	_bEnable: 					BOOL;
	
	_bManual:                   BOOL;//屏蔽取uc
	
	_TakeUcCheck0FTrig:         Tc2_Standard.F_TRIG;
	
END_VAR

_station REF= G_arrStation[E_Station.TakeUc];
_station.arrName[E_Language.Chinese]:="取Uc站";
_station.arrName[E_Language.Vietnamese]:="Lấy ga";
_bEnable:=NOT GVL.stSetting.arrStationShield[E_Station.TakeUc];

IF GVL_Data.stRecipe.eMachineType=E_MachineType._311 THEN
	A_Home311();
	A_Auto311();
ELSE
	A_Home();
	A_Auto();
END_IF

_bManual:=FALSE;//屏蔽取UC

_TakeUcCheck0FTrig(CLK:= GVL.I.bTakeUcCheck0, Q=> );

GVL._arrAutoTimer[E_Timer.OpenLockCheckF](IN:=NOT GVL.I.bOpenLockCheck AND GVL.I.bOpenLockLift_Cyl_H, PT:=TO_TIME(GVL_Data.stRecipe.arrAutoTon[E_Timer.OpenLockCheckF]), Q=>GVL._arrAutoTimerOut[E_Timer.OpenLockCheckF] , ET=> );

ACTION A_Auto:
CASE _station.iStepNow OF
	1000:
		_station.arrInfo[E_Language.Chinese]:="初始化完成等待启动";
		IF _bEnable THEN
			_station.iStepNext:=1101;
		END_IF
	1101:
		_station.arrInfo[E_Language.Chinese]:="判断是否有料";
		IF NOT GVL.I.bTakeUcCheck1 THEN
			_station.iStepNext:=1201;
		END_IF
	1201:
		_station.arrInfo[E_Language.Chinese]:="请求放料";
		GVL.stHandshake.bTakeUcToOpen:=TRUE;
		IF GVL.stHandshake.bOpenToTakeUc THEN
			_station.iStepNext:=1301;
		END_IF
	1301://安装了取UC站流入传感器但未移至阻挡气缸后侧的启用此条
		_station.arrInfo[E_Language.Chinese]:="等待产品从解锁站流出";
		GVL.stOverTime.bTakeUcCheck1:=TRUE;
		IF GVL.I.bTakeUcCheck1 OR GVL.I.bTakeUcCheck0 THEN  				
			GVL.stOverTime.bTakeUcCheck1:=FALSE;
			_station.iStepNext:=1401;
		END_IF  
		
(*	1301://未安装了取UC站流入传感器的启用此条
		_station.arrInfo[E_Language.Chinese]:="等待产品从解锁站流出";
		GVL.stOverTime.bTakeUcCheck1:=TRUE;
		IF GVL._arrAutoTimerOut[E_Timer.OpenLockCheckF] THEN  				
			GVL.stOverTime.bTakeUcCheck1:=FALSE;
			_station.iStepNext:=1401;
		END_IF*)
		
		
(*	1301://安装了取UC站流入传感器并且移至阻挡气缸后侧的启用此条
		_station.arrInfo[E_Language.Chinese]:="等待产品从解锁站流出";
		GVL.stOverTime.bTakeUcCheck1:=TRUE;
		IF NOT GVL.I.bOpenLockCheck THEN  				
			GVL.stOverTime.bTakeUcCheck1:=FALSE;
			_station.iStepNext:=1311;
		END_IF		
	1311:		
		_station.arrInfo[E_Language.Chinese]:="产品从解锁站流出确认";
		IF _TakeUcCheck0FTrig.Q THEN
			_station.iStepNext:=1401;
		END_IF	*)	
		
		
	1401:
		_station.arrInfo[E_Language.Chinese]:="复位请求信号";
		GVL.stHandshake.bTakeUcToOpen:=FALSE;
		IF NOT GVL.stHandshake.bOpenToTakeUc THEN
			_station.iStepNext:=1411;
		END_IF
	1411:
		_station.arrInfo[E_Language.Chinese]:="等待产品到位";
		GVL.stOverTime.bTakeUcCheck1:=TRUE;
		IF GVL.I.bTakeUcCheck1 THEN
			GVL.stOverTime.bTakeUcCheck1:=FALSE;
			_station.iStepNext:=1501;
		END_IF			
	1501:
		_station.arrInfo[E_Language.Chinese]:="顶升气缸伸出";	
		IF G_arrFbCylinder[E_Cylinder.TakeUcLift].M_WorkRequest() THEN
			_station.iStepNext:=1511;
		END_IF
	1511:
		_station.arrInfo[E_Language.Chinese]:="夹紧气缸夹紧 阻挡气缸缩回";
        IF M_ClampWork() AND G_arrFbCylinder[E_Cylinder.TakeUcPrevent].M_HomeRequest() THEN
			_station.iStepNext:=SEL(GVL_Data.stRecipe.eMachineType=E_MachineType._373,1521,1512);
		END_IF
	1512:		
		_station.arrInfo[E_Language.Chinese]:="判断工装有无误合盖";
		IF GVL.I.bFrockCloseCheck OR GVL.stSetting.bFrockCloseCheckShield THEN
			_station.iStepNext:=1521;
		ELSE
			_station.iStepNext:=2301;
		END_IF	
	1521:
		_station.arrInfo[E_Language.Chinese]:="校平气缸伸出";
	   	IF  M_StandardWork() THEN
			_station.iStepNext:=SEL(_bManual,1601,1751);
		END_IF
	1601:
		_station.arrInfo[E_Language.Chinese]:="请求取UC";
		GVL.stHandshake.bTakeUcToTakeUc_M:=TRUE;
		IF  GVL.stHandshake.bTakeUc_MToTakeUc THEN
			_station.iStepNext:=1651;
		END_IF
	1651:
		CASE GVL_Data.stRecipe.eMachineType OF
			E_MachineType._069,E_MachineType._200:
				_station.arrInfo[E_Language.Chinese]:="侧推气缸伸出";
				IF G_arrFbCylinder[E_Cylinder.TakeUcPush].M_WorkRequest() THEN
					_station.iStepNext:=1701;
				END_IF
			ELSE
				_station.iStepNext:=1701;
		END_CASE
	1701:
		_station.arrInfo[E_Language.Chinese]:="复位请求信号";
		GVL.stHandshake.bTakeUcToTakeUc_M:=FALSE;
		IF NOT  GVL.stHandshake.bTakeUc_MToTakeUc THEN
			_station.iStepNext:=1751;
		END_IF
	1751:
		_station.arrInfo[E_Language.Chinese]:="校平气缸缩回";
		IF M_StandardHome()  THEN
			_station.iStepNext:=1801;
		END_IF
	1801:
		_station.arrInfo[E_Language.Chinese]:="侧推气缸伸出";
		IF G_arrFbCylinder[E_Cylinder.TakeUcPush].M_WorkRequest() THEN
			_station.iStepNext:=1901;
		END_IF
	1901:
		_station.arrInfo[E_Language.Chinese]:="旋转气缸至左位";
		IF G_arrFbCylinder[E_Cylinder.TakeUcRotate].M_HomeRequest() THEN
			_station.iStepNext:=2001;
		END_IF		
	2001:
		_station.arrInfo[E_Language.Chinese]:="侧推气缸复位 夹紧气缸松开";
		IF G_arrFbCylinder[E_Cylinder.TakeUcPush].M_HomeRequest() AND M_ClampHome() THEN
			_station.iStepNext:=2301;
		END_IF
	2301:
		_station.arrInfo[E_Language.Chinese]:="等待下工工装站请求放料";
		IF GVL.stHandshake.bUnloadFrockToTakeUc THEN
			GVL.stHandshake.bTakeUcToUnloadFrock:=TRUE;
			GVL.stHandshake.bTakeUcToOpen:=TRUE;//同时请求解锁站放料
			_station.iStepNext:=2401;
		END_IF
	2401:
		_station.arrInfo[E_Language.Chinese]:="顶升气缸缩回,旋转气缸至右位";
		IF G_arrFbCylinder[E_Cylinder.TakeUcLift].M_HomeRequest() AND G_arrFbCylinder[E_Cylinder.TakeUcRotate].M_WorkRequest() THEN	
            _station.iStepNext:=2501;
		END_IF
	2501:
		_station.arrInfo[E_Language.Chinese]:="等待复位请求放料";
		IF NOT GVL.stHandshake.bUnloadFrockToTakeUc THEN
			GVL.stHandshake.bTakeUcToUnloadFrock:=FALSE;
			_station.iStepNext:=2601;
		END_IF	
	2601:
		_station.arrInfo[E_Language.Chinese]:="阻挡气缸伸出";
		IF G_arrFbCylinder[E_Cylinder.TakeUcPrevent].M_WorkRequest() THEN
			_station.iStepNext:=1201;
		END_IF	

END_CASE
END_ACTION

ACTION A_Auto311:
CASE _station.iStepNow OF
	1000:
		_station.arrInfo[E_Language.Chinese]:="初始化完成等待启动";
		IF _bEnable THEN
			_station.iStepNext:=1101;
		END_IF
	1101:
		_station.arrInfo[E_Language.Chinese]:="判断是否有料";
		IF NOT GVL.I.bTakeUcCheck1 THEN
			_station.iStepNext:=1201;
		END_IF
	1201:
		_station.arrInfo[E_Language.Chinese]:="请求放料";
		GVL.stHandshake.bTakeUcToOpen:=TRUE;
		IF GVL.stHandshake.bOpenToTakeUc THEN
			_station.iStepNext:=1301;
		END_IF
	1301://安装了取UC站流入传感器但未移至阻挡气缸后侧的启用此条
		_station.arrInfo[E_Language.Chinese]:="等待产品从解锁站流出";
		GVL.stOverTime.bTakeUcCheck1:=TRUE;
		IF GVL.I.bTakeUcCheck1 OR GVL.I.bTakeUcCheck0 THEN  				
			GVL.stOverTime.bTakeUcCheck1:=FALSE;
			_station.iStepNext:=1401;
		END_IF  
		
(*	1301://未安装了取UC站流入传感器的启用此条
		_station.arrInfo[E_Language.Chinese]:="等待产品从解锁站流出";
		GVL.stOverTime.bTakeUcCheck1:=TRUE;
		IF GVL._arrAutoTimerOut[E_Timer.OpenLockCheckF] THEN  				
			GVL.stOverTime.bTakeUcCheck1:=FALSE;
			_station.iStepNext:=1401;
		END_IF  *)
		
		
(*	1301://安装了取UC站流入传感器并且移至阻挡气缸后侧的启用此条
		_station.arrInfo[E_Language.Chinese]:="等待产品从解锁站流出";
		GVL.stOverTime.bTakeUcCheck1:=TRUE;
		IF NOT GVL.I.bOpenLockCheck THEN  				
			GVL.stOverTime.bTakeUcCheck1:=FALSE;
			_station.iStepNext:=1311;
		END_IF		
	1311:		
		_station.arrInfo[E_Language.Chinese]:="产品从解锁站流出确认";
		IF _TakeUcCheck0FTrig.Q THEN
			_station.iStepNext:=1401;
		END_IF	*)		
	1401:
		_station.arrInfo[E_Language.Chinese]:="复位请求信号";
		GVL.stHandshake.bTakeUcToOpen:=FALSE;
		IF NOT GVL.stHandshake.bOpenToTakeUc THEN
			_station.iStepNext:=1411;
		END_IF
	1411:
		_station.arrInfo[E_Language.Chinese]:="等待产品到位";
		GVL.stOverTime.bTakeUcCheck1:=TRUE;
		IF GVL.I.bTakeUcCheck1 THEN
			
			IF GVL.TakeUcSafeCheckNG_OpenLock THEN
				GVL.TakeUcSafeCheckNG_TakeUc:=TRUE;
			ELSE
				GVL.TakeUcSafeCheckNG_TakeUc:=FALSE;	
			END_IF	
			
			GVL.stOverTime.bTakeUcCheck1:=FALSE;
			_station.iStepNext:=1501;
		END_IF				
	1501:
		_station.arrInfo[E_Language.Chinese]:="顶升气缸伸出";
		IF G_arrFbCylinder[E_Cylinder.TakeUcLift].M_WorkRequest() THEN
			_station.iStepNext:=1502;
		END_IF
	1502:		
		_station.arrInfo[E_Language.Chinese]:="检测工装有无误合盖";
		IF NOT GVL.TakeUcSafeCheckNG_TakeUc THEN
			_station.iStepNext:=1511;
		ELSE
			_station.iStepNext:=1503;
		END_IF
	1503:
		_station.arrInfo[E_Language.Chinese]:="侧推气缸伸出";
		GVL.TakeUcSafeCheckNG_TakeUc:=FALSE;
		IF  NOT GVL.TakeUcSafeCheckNG_TakeUc THEN
			_station.iStepNext:=2201;
		END_IF	
	1511:
		_station.arrInfo[E_Language.Chinese]:="请求取UC";
		GVL.stHandshake.bTakeUcToTakeUc_M:=TRUE;
		IF  GVL.stHandshake.bTakeUc_MToTakeUc THEN
			_station.iStepNext:=1551;
		END_IF	
	1551:
		_station.arrInfo[E_Language.Chinese]:="侧推气缸伸出 侧推气缸1伸出";
		IF  G_arrFbCylinder[E_Cylinder.TakeUcPush].M_WorkRequest() AND G_arrFbCylinder[E_Cylinder.TakeUcPush1].M_WorkRequest() THEN
			_station.iStepNext:=1601;
		END_IF
	1601:
		_station.arrInfo[E_Language.Chinese]:="阻挡气缸缩回 升降气缸伸出";
		IF  G_arrFbCylinder[E_Cylinder.TakeUcPrevent].M_HomeRequest() AND G_arrFbCylinder[E_Cylinder.TakeUcElevator].M_WorkRequest() THEN
			_station.iStepNext:=1611;
		END_IF
	1611:
		 IF NOT _bManual  THEN
			_station.iStepNext:=1621;
			ELSE
			_station.iStepNext:=1801;
		END_IF
	1621:
		_station.arrInfo[E_Language.Chinese]:="复位请求信号";
		GVL.stHandshake.bTakeUcToTakeUc_M:=FALSE;
		IF NOT  GVL.stHandshake.bTakeUc_MToTakeUc THEN
			_station.iStepNext:=1651;
		END_IF
	1651:
		_station.arrInfo[E_Language.Chinese]:="请求取UC2";
		GVL.stHandshake.bTakeUcToTakeUc_M_2:=TRUE;
		IF  GVL.stHandshake.bTakeUc_MToTakeUc_2 THEN
			_station.iStepNext:=1701;
		END_IF
	1701:
		_station.arrInfo[E_Language.Chinese]:="复位请求信号2";
		GVL.stHandshake.bTakeUcToTakeUc_M_2:=FALSE;
		IF NOT  GVL.stHandshake.bTakeUc_MToTakeUc_2 THEN
			_station.iStepNext:=1801;
		END_IF
	1801:
		_station.arrInfo[E_Language.Chinese]:="旋转气缸至右位 侧推1缩回";
		IF G_arrFbCylinder[E_Cylinder.TakeUcRotate].M_WorkRequest() AND G_arrFbCylinder[E_Cylinder.TakeUcPush1].M_HomeRequest() THEN
			_station.iStepNext:=1901;
		END_IF
	1901:
		_station.arrInfo[E_Language.Chinese]:="侧推气缸复位 升降气缸缩回";
		IF G_arrFbCylinder[E_Cylinder.TakeUcPush].M_HomeRequest() AND G_arrFbCylinder[E_Cylinder.TakeUcElevator].M_HomeRequest() THEN
			_station.iStepNext:=2201;
		END_IF
(*	2001:
		_station.arrInfo[E_Language.Chinese]:="阻挡气缸缩回";
		IF  G_arrFbCylinder[E_Cylinder.TakeUcPrevent].M_HomeRequest() THEN
			_station.iStepNext:=2201;
		END_IF*)
	2201:
		_station.arrInfo[E_Language.Chinese]:="等待下工工装站请求放料";
		IF GVL.stHandshake.bUnloadFrockToTakeUc THEN
			GVL.stHandshake.bTakeUcToUnloadFrock:=TRUE;
			GVL.stHandshake.bTakeUcToOpen:=TRUE;//同时请求解锁站放料
			_station.iStepNext:=2301;
		END_IF
	2301:
		_station.arrInfo[E_Language.Chinese]:="顶升气缸缩回 旋转气缸复位 阻挡气缸缩回";
		IF G_arrFbCylinder[E_Cylinder.TakeUcLift].M_HomeRequest()  AND G_arrFbCylinder[E_Cylinder.TakeUcRotate].M_HomeRequest() AND G_arrFbCylinder[E_Cylinder.TakeUcPrevent].M_HomeRequest() THEN
			_station.iStepNext:=2401;
		END_IF
	2401:
		_station.arrInfo[E_Language.Chinese]:="等待复位请求放料";
		IF NOT GVL.stHandshake.bUnloadFrockToTakeUc THEN
			GVL.stHandshake.bTakeUcToUnloadFrock:=FALSE;
			_station.iStepNext:=2601;
		END_IF		
	2601:
		_station.arrInfo[E_Language.Chinese]:="阻挡气缸伸出";
		IF G_arrFbCylinder[E_Cylinder.TakeUcPrevent].M_WorkRequest() THEN
			_station.iStepNext:=1201;
		END_IF	

END_CASE
END_ACTION

ACTION A_Home:
CASE _station.iStepNow OF
	0:
		_station.arrInfo[E_Language.Chinese]:="等待初始化";
		_station.iStepNext:=SEL(_bEnable,1000,100);;
	100:
		IF GVL.I.bTakeUc1Y_Cyl_W THEN  //确认取UC模组在初始位时再开始初始化
			_station.iStepNext:=110;
		END_IF
	110:	
		_station.arrInfo[E_Language.Chinese]:="侧推气缸缩回";
		IF G_arrFbCylinder[E_Cylinder.TakeUcPush].M_HomeRequest() THEN
			_station.iStepNext:=200;
		END_IF
	200:
		_station.arrInfo[E_Language.Chinese]:="旋转气缸至右位";
		IF G_arrFbCylinder[E_Cylinder.TakeUcRotate].M_WorkRequest() THEN
			_station.iStepNext:=300;
		END_IF
	300:
		_station.arrInfo[E_Language.Chinese]:="校平气缸缩回";
		IF M_StandardHome() THEN
			_station.iStepNext:=400;
		END_IF
	400:
	    _station.arrInfo[E_Language.Chinese]:="夹紧气缸松开";
		IF M_ClampHome() THEN
			_station.iStepNext:=500;
		END_IF
	500:
	    _station.arrInfo[E_Language.Chinese]:="顶升气缸缩回";
		IF G_arrFbCylinder[E_Cylinder.TakeUcLift].M_HomeRequest() THEN
			_station.iStepNext:=600;
		END_IF
	600:
		_station.arrInfo[E_Language.Chinese]:="阻挡气缸伸出";
		IF G_arrFbCylinder[E_Cylinder.TakeUcPrevent].M_WorkRequest() THEN
			_station.iStepNext:=1000;
		END_IF
		
		
		
		
END_CASE
END_ACTION

ACTION A_Home311:
CASE _station.iStepNow OF
	0:
		_station.arrInfo[E_Language.Chinese]:="等待初始化";
		_station.iStepNext:=SEL(_bEnable,1000,100);;
	100:
		IF GVL.I.bTakeUc1Y_Cyl_W THEN  //确认取UC模组在初始位时再开始初始化
			_station.iStepNext:=110;
		END_IF			
	110:
		_station.arrInfo[E_Language.Chinese]:="升降气缸缩回";
		IF G_arrFbCylinder[E_Cylinder.TakeUcElevator].M_HomeRequest() THEN
			_station.iStepNext:=150;
		END_IF
	150:
		_station.arrInfo[E_Language.Chinese]:="侧推气缸缩回";
		IF G_arrFbCylinder[E_Cylinder.TakeUcPush].M_HomeRequest() AND G_arrFbCylinder[E_Cylinder.TakeUcPush1].M_HomeRequest()  THEN
			_station.iStepNext:=200;
		END_IF
	200:
		_station.arrInfo[E_Language.Chinese]:="旋转气缸至左位";
		IF G_arrFbCylinder[E_Cylinder.TakeUcRotate].M_HomeRequest() THEN
			_station.iStepNext:=300;
		END_IF
	300:
		_station.arrInfo[E_Language.Chinese]:="阻挡气缸伸出";
		IF G_arrFbCylinder[E_Cylinder.TakeUcPrevent].M_WorkRequest() THEN
			_station.iStepNext:=400;
		END_IF
	400:
		_station.arrInfo[E_Language.Chinese]:="顶升气缸缩回";
		IF G_arrFbCylinder[E_Cylinder.TakeUcLift].M_HomeRequest() THEN
			_station.iStepNext:=1000;
		END_IF
END_CASE
END_ACTION

METHOD M_ClampHome : BOOL
VAR_INPUT
END_VAR
CASE GVL_Data.stRecipe.eMachineType OF
	E_MachineType._367:
		M_ClampHome:=G_arrFbCylinder[E_Cylinder.TakeUcFrockClamp].M_HomeRequest();
	ELSE
		M_ClampHome:=TRUE;
END_CASE
END_METHOD

METHOD M_ClampWork : BOOL
VAR_INPUT
END_VAR
CASE GVL_Data.stRecipe.eMachineType OF
	E_MachineType._367:
		M_ClampWork:=G_arrFbCylinder[E_Cylinder.TakeUcFrockClamp].M_WorkRequest();
	ELSE
		M_ClampWork:=TRUE;
END_CASE
END_METHOD

METHOD M_StandardHome : BOOL
VAR_INPUT
END_VAR
CASE GVL_Data.stRecipe.eMachineType OF
	E_MachineType._367:
		M_StandardHome:=G_arrFbCylinder[E_Cylinder.TakeUcStandard].M_HomeRequest();
	ELSE
		M_StandardHome:=TRUE;
END_CASE
END_METHOD

METHOD M_StandardWork : BOOL
VAR_INPUT
END_VAR
CASE GVL_Data.stRecipe.eMachineType OF
	E_MachineType._367:
		M_StandardWork:=G_arrFbCylinder[E_Cylinder.TakeUcStandard].M_WorkRequest();
	ELSE
		M_StandardWork:=TRUE;
END_CASE
END_METHOD

END_PROGRAM

// ---- POUs/P_StationTakeUc_M.TcPOU
PROGRAM P_StationTakeUc_M
VAR
	_station:					REFERENCE TO ST_SystemStation;
	_bEnable: 					BOOL;
	
	_ton:                       ARRAY [0..20] OF TON;;
	_frig:                      ARRAY [0..20] OF R_TRIG;

	RLSE: INT;
END_VAR

_station REF= G_arrStation[E_Station.TakeUc_M];
_station.arrName[E_Language.Chinese]:="取Uc模组";
_station.arrName[E_Language.Vietnamese]:="Lấy mô-đun Uc";
_bEnable:=NOT GVL.stSetting.arrStationShield[E_Station.TakeUc_M];
A_Auto();
A_Home();

ACTION A_Auto:
CASE _station.iStepNow OF
	1000:
		_station.arrInfo[E_Language.Chinese]:="初始化完成等待启动";
		IF _bEnable THEN
			_station.iStepNext:=1101;
		END_IF
	1101:
			_station.arrInfo[E_Language.Chinese]:="Z模组至取Uc位";
		IF GVL_Data.stRecipe.eMachineType=E_MachineType._367 THEN
			IF M_ZTakeUc() THEN
				_station.iStepNext:=1111;
			END_IF
		ELSE
			_station.iStepNext:=1111;
		END_IF
	1111:
		_station.arrInfo[E_Language.Chinese]:="等待取Uc站请求取料1";
		IF GVL.stHandshake.bTakeUcToTakeUc_M THEN
			 GVL.stHandshake.bTakeUc_MToTakeUc:=TRUE;
			 _station.iStepNext:=1151;
		END_IF	
	1151:
	    _station.arrInfo[E_Language.Chinese]:="Y气缸至前位";
		IF G_arrFbCylinder[E_Cylinder.TakeUc1Y].M_HomeRequest()THEN
			_station.iStepNext:=SEL(GVL_Data.stRecipe.eMachineType=E_MachineType._311,1201,1161);			
		END_IF	
	1161:	
		_station.arrInfo[E_Language.Chinese]:="等待复位取Uc请求1";
		IF NOT  GVL.stHandshake.bTakeUcToTakeUc_M THEN
			 GVL.stHandshake.bTakeUc_MToTakeUc:=FALSE;			
			 _station.iStepNext:=1171;				 
		END_IF 
		
	1171:
		_station.arrInfo[E_Language.Chinese]:="等待取Uc站请求取料2";
		IF GVL.stHandshake.bTakeUcToTakeUc_M_2 THEN
			 GVL.stHandshake.bTakeUc_MToTakeUc_2:=TRUE;
			 _station.iStepNext:=1201;
		END_IF	
		
